// TwinCAT 3 PLC project CNM_AssertionInterfaceLib
// Title: CNM_AssertionInterfaces
// Company: ekvip automation GmbH
// Author: elfrosch
// ProjectVersion: 0.1.1.0
// Description: This library provides an abstract class `AbstractAssertor` to ease assert statements. It provides assert statements in a [fluent interface](https://en.wikipedia.org/wiki/Fluent_interface) style for the most common data types. .. <legal notes> legal notes ================= | SPDX-FileCopyrightText: © 2022 ekvip automation GmbH <info@ekvip.de> | SPDX-License-Identifier: Apache-2.0 | For details check: Apache-2.0_ .. _Apache-2.0: https://www.apache.org/licenses/LICENSE-2.0 .. </legal notes>
// ProgramVersion: 3.1.4026.19
// libraries:
//   CNM_AbstractObject, * (ekvip automation GmbH)
//   CNM_ReturnTypes, * (ekvip automation GmbH)
//   CNM_UnicodeUtilities, * (ekvip automation GmbH)
//   SysMem, * (System)
//   Tc2_Standard, * (Beckhoff Automation GmbH)
//   Tc2_System, * (Beckhoff Automation GmbH)
//   Tc2_Utilities, * (Beckhoff Automation GmbH)
// project tree:
//   Assertor/Assertions/BinaryAssertions/classes/ BinaryAssertions.TcPOU
//   Assertor/Assertions/BinaryAssertions/interfaces/ IBinaryAssertions.TcIO
//   Assertor/Assertions/BitNumberAssertions/Byte/classes/ ByteAssertions.TcPOU
//   Assertor/Assertions/BitNumberAssertions/Byte/interfaces/ IByteAssertions.TcIO
//   Assertor/Assertions/BitNumberAssertions/Byte/types/subranges/ BitNumberByte.TcDUT
//   Assertor/Assertions/BitNumberAssertions/classes/ BitNumberAssertions.TcPOU
//   Assertor/Assertions/BitNumberAssertions/Dword/classes/ DWordAssertions.TcPOU
//   Assertor/Assertions/BitNumberAssertions/Dword/interfaces/ IDwordAssertions.TcIO
//   Assertor/Assertions/BitNumberAssertions/Dword/types/subranges/ BitNumberDWord.TcDUT
//   Assertor/Assertions/BitNumberAssertions/interfaces/ IBitNumberAssertions.TcIO
//   Assertor/Assertions/BitNumberAssertions/Lword/classes/ LWordAssertions.TcPOU
//   Assertor/Assertions/BitNumberAssertions/Lword/interfaces/ ILwordAssertions.TcIO
//   Assertor/Assertions/BitNumberAssertions/Lword/types/subranges/ BitNumberLWord.TcDUT
//   Assertor/Assertions/BitNumberAssertions/Word/classes/ WordAssertions.TcPOU
//   Assertor/Assertions/BitNumberAssertions/Word/interfaces/ IWordAssertions.TcIO
//   Assertor/Assertions/BitNumberAssertions/Word/types/subranges/ BitNumberWord.TcDUT
//   Assertor/Assertions/BitNumberAssertions/XWord/classes/ XWordAssertions.TcPOU
//   Assertor/Assertions/BitNumberAssertions/XWord/interfaces/ IXWordAssertions.TcIO
//   Assertor/Assertions/BitNumberAssertions/XWord/types/subranges/ BitNumberXWord.TcDUT
//   Assertor/Assertions/BooleanAssertion/classes/ BooleanAssertion.TcPOU
//   Assertor/Assertions/BooleanAssertion/interfaces/ IBooleanAssertion.TcIO
//   Assertor/Assertions/classes/ Assertions.TcPOU
//   Assertor/Assertions/DateAndTimeAssertions/32Bit/classes/ SimpleDateAndTimeAssertions.TcPOU
//   Assertor/Assertions/DateAndTimeAssertions/32Bit/Date/classes/ DateAssertions32Bit.TcPOU
//   Assertor/Assertions/DateAndTimeAssertions/32Bit/Date/interfaces/ I32BitDateAssertions.TcIO
//   Assertor/Assertions/DateAndTimeAssertions/32Bit/DT/classes/ DateTimeAssertions32Bit.TcPOU
//   Assertor/Assertions/DateAndTimeAssertions/32Bit/DT/interfaces/ I32BitDtAssertions.TcIO
//   Assertor/Assertions/DateAndTimeAssertions/32Bit/interfaces/ ISimpleDateAndTimeAssertions.TcIO
//   Assertor/Assertions/DateAndTimeAssertions/32Bit/TOD/classes/ TimeOfDayAssertions32Bit.TcPOU
//   Assertor/Assertions/DateAndTimeAssertions/32Bit/TOD/interfaces/ I32BitTodAssertions.TcIO
//   Assertor/Assertions/DateAndTimeAssertions/64Bit/classes/ LongDateAndTimeAssertions.TcPOU
//   Assertor/Assertions/DateAndTimeAssertions/64Bit/LDate/classes/ DateAssertions64Bit.TcPOU
//   Assertor/Assertions/DateAndTimeAssertions/64Bit/LDate/interfaces/ I64BitDateAssertions.TcIO
//   Assertor/Assertions/DateAndTimeAssertions/64Bit/LDT/classes/ DateTimeAssertions64Bit.TcPOU
//   Assertor/Assertions/DateAndTimeAssertions/64Bit/LDT/interfaces/ I64BitDtAssertions.TcIO
//   Assertor/Assertions/DateAndTimeAssertions/64Bit/interfaces/ ILongDateAndTimeAssertions.TcIO
//   Assertor/Assertions/DateAndTimeAssertions/64Bit/LTOD/classes/ TimeOfDayAssertions64Bit.TcPOU
//   Assertor/Assertions/DateAndTimeAssertions/64Bit/LTOD/interfaces/ I64BitTodAssertions.TcIO
//   Assertor/Assertions/DateAndTimeAssertions/classes/ DateAndTimeAssertions.TcPOU
//   Assertor/Assertions/DateAndTimeAssertions/interfaces/ IDateAndTimeAssertions.TcIO
//   Assertor/Assertions/FloatAssertions/classes/ FloatAssertions.TcPOU
//   Assertor/Assertions/FloatAssertions/interfaces/ IFloatAssertions.TcIO
//   Assertor/Assertions/FloatAssertions/Lreal/classes/ LrealAssertions.TcPOU
//   Assertor/Assertions/FloatAssertions/Lreal/interfaces/ ILrealAssertions.TcIO
//   Assertor/Assertions/FloatAssertions/Real/classes/ RealAssertions.TcPOU
//   Assertor/Assertions/FloatAssertions/Real/interfaces/ IRealAssertions.TcIO
//   Assertor/Assertions/IntegerAssertions/classes/ IntegerAssertions.TcPOU
//   Assertor/Assertions/IntegerAssertions/interfaces/ IIntegerAssertions.TcIO
//   Assertor/Assertions/IntegerAssertions/signed/classes/ SignedIntegerAssertions.TcPOU
//   Assertor/Assertions/IntegerAssertions/signed/Dint/classes/ DintAssertions.TcPOU
//   Assertor/Assertions/IntegerAssertions/signed/Dint/interfaces/ IDintAssertions.TcIO
//   Assertor/Assertions/IntegerAssertions/signed/interfaces/ ISignedIntegerAssertions.TcIO
//   Assertor/Assertions/IntegerAssertions/signed/Int/classes/ IntAssertions.TcPOU
//   Assertor/Assertions/IntegerAssertions/signed/Int/interfaces/ IIntAssertions.TcIO
//   Assertor/Assertions/IntegerAssertions/signed/Lint/classes/ LintAssertions.TcPOU
//   Assertor/Assertions/IntegerAssertions/signed/Lint/interfaces/ ILintAssertions.TcIO
//   Assertor/Assertions/IntegerAssertions/signed/Sint/classes/ SintAssertions.TcPOU
//   Assertor/Assertions/IntegerAssertions/signed/Sint/interfaces/ ISintAssertions.TcIO
//   Assertor/Assertions/IntegerAssertions/signed/Xint/classes/ XintAssertions.TcPOU
//   Assertor/Assertions/IntegerAssertions/signed/Xint/interfaces/ IXintAssertions.TcIO
//   Assertor/Assertions/IntegerAssertions/unsigned/classes/ UnsignedIntegerAssertions.TcPOU
//   Assertor/Assertions/IntegerAssertions/unsigned/interfaces/ IUnsignedIntegerAssertions.TcIO
//   Assertor/Assertions/IntegerAssertions/unsigned/Udint/classes/ UdintAssertions.TcPOU
//   Assertor/Assertions/IntegerAssertions/unsigned/Udint/interfaces/ IUdintAssertions.TcIO
//   Assertor/Assertions/IntegerAssertions/unsigned/Uint/classes/ UintAssertions.TcPOU
//   Assertor/Assertions/IntegerAssertions/unsigned/Uint/interfaces/ IUintAssertions.TcIO
//   Assertor/Assertions/IntegerAssertions/unsigned/Ulint/classes/ UlintAssertions.TcPOU
//   Assertor/Assertions/IntegerAssertions/unsigned/Ulint/interfaces/ IUlintAssertions.TcIO
//   Assertor/Assertions/IntegerAssertions/unsigned/Usint/classes/ UsintAssertions.TcPOU
//   Assertor/Assertions/IntegerAssertions/unsigned/Usint/interfaces/ IUsintAssertions.TcIO
//   Assertor/Assertions/IntegerAssertions/unsigned/Uxint/classes/ UxintAssertions.TcPOU
//   Assertor/Assertions/IntegerAssertions/unsigned/Uxint/interfaces/ IUxintAssertions.TcIO
//   Assertor/Assertions/interfaces/ IAssertions.TcIO
//   Assertor/Assertions/ObjectAssertions/classes/ ObjectAssertions.TcPOU
//   Assertor/Assertions/ObjectAssertions/interfaces/ IObjectAssertions.TcIO
//   Assertor/Assertions/PointerAssertions/classes/ PointerAssertions.TcPOU
//   Assertor/Assertions/PointerAssertions/interfaces/ IPointerAssertions.TcIO
//   Assertor/Assertions/StringAssertion/classes/ AbstractStringPointerAssertions.TcPOU, StringAssertions.TcPOU
//   Assertor/Assertions/StringAssertion/interfaces/ IStringAssertions.TcIO
//   Assertor/Assertions/StringAssertion/Win125x/classes/ Windows125xStringAssertions.TcPOU, Windows125xStringPointerAssertions.TcPOU
//   Assertor/Assertions/StringAssertion/Win125x/interfaces/ IWindows125xStringAssertions.TcIO, IWindows125xStringPointerAssertions.TcIO
//   Assertor/Assertions/StringAssertion/Unicode/Classes/ UnicodeAssertions.TcPOU
//   Assertor/Assertions/StringAssertion/Unicode/Classes/UTF-16/ Utf16StringAssertions.TcPOU, Utf16StringPointerAssertions.TcPOU
//   Assertor/Assertions/StringAssertion/Unicode/Classes/UTF-8/ Utf8StringAssertions.TcPOU, Utf8StringPointerAssertions.TcPOU
//   Assertor/Assertions/StringAssertion/Unicode/enumerations/ UnicodeStringLengthUnit.TcDUT
//   Assertor/Assertions/StringAssertion/Unicode/Interfaces/ IUnicodeStringAssertions.TcIO
//   Assertor/Assertions/StringAssertion/Unicode/Interfaces/UTF-16/ IUtf16StringAssertions.TcIO, IUtf16StringPointerAssertions.TcIO
//   Assertor/Assertions/StringAssertion/Unicode/Interfaces/UTF-8/ IUtf8StringAssertions.TcIO, IUtf8StringPointerAssertions.TcIO
//   Assertor/Assertions/TimeAssertions/classes/ TimeAssertions.TcPOU
//   Assertor/Assertions/TimeAssertions/interfaces/ ITimeAssertions.TcIO
//   Assertor/Assertions/TimeAssertions/LTime/classes/ LongTimeAssertions.TcPOU
//   Assertor/Assertions/TimeAssertions/LTime/interfaces/ I64BitTimeAssertions.TcIO
//   Assertor/Assertions/TimeAssertions/Time/classes/ SimpleTimeAssertions.TcPOU
//   Assertor/Assertions/TimeAssertions/Time/interfaces/ I32BitTimeAssertions.TcIO
//   Assertor/classes/ AbstractAssertion.TcPOU, AbstractAssertor.TcPOU
//   Assertor/interfaces/ IAssertor.TcIO, IAssertCallBack.TcIO, IAssertCallBackSetter.TcIO
//   Assertor/types/aliases/ AssertMessage.TcDUT
//   Project Information/ F_GetCompany.TcPOU, F_GetTitle.TcPOU, F_GetVersion.TcPOU
//   Version/ Global_Version.TcGVL
// real-time tasks:
//   TASK CNC-Task ADS: cycle default, priority 7, ADS port 558
//   TASK CNC-Task COM: cycle T#10ms, priority 13, ADS port 556
//   TASK CNC-Task SDA: cycle T#10ms, priority 8, ADS port 555
//   TASK CNC-Task GEO: cycle T#2ms, priority 3, ADS port 554

// ---- Assertor/Assertions/BitNumberAssertions/Byte/types/subranges/BitNumberByte.TcDUT
(*

## Short summary

BitNumberByte is an alias of ``USINT(0..7)``.
This data type exists so that no one can provoke an overflow of the bit numbers.
It's used as parameter at 
`IByteAssertions.bitXIsEqualTo` 
`IByteAssertions.bitXIsNotEqualTo` 
`IByteAssertions.bitXIsSet` 
`IByteAssertions.bitXIsUnset` 

.. <legal notes>

legal notes
=================
| SPDX-FileCopyrightText: © 2022 ekvip automation GmbH <info@ekvip.de>
| SPDX-License-Identifier: Apache-2.0
| For details check: Apache-2.0_

.. _Apache-2.0: https://www.apache.org/licenses/LICENSE-2.0

.. </legal notes>

*)

TYPE
	BitNumberByte :USINT(0..7); 
END_TYPE

// ---- Assertor/Assertions/BitNumberAssertions/Dword/types/subranges/BitNumberDWord.TcDUT
(*

## Short summary

 BitNumberDWord is an alias of ``USINT(0..31)``.
 This data type exists so that no one can provoke an overflow of the bit numbers.
 It's used as parameter of 
 `IDwordAssertions.bitXIsEqualTo` 
 `IDwordAssertions.bitXIsNotEqualTo` 
 `IDwordAssertions.bitXIsSet` 
 `IDwordAssertions.bitXIsUnset` 

.. <legal notes>

legal notes
=================
| SPDX-FileCopyrightText: © 2022 ekvip automation GmbH <info@ekvip.de>
| SPDX-License-Identifier: Apache-2.0
| For details check: Apache-2.0_

.. _Apache-2.0: https://www.apache.org/licenses/LICENSE-2.0

.. </legal notes>

*)

TYPE
	BitNumberDWord :USINT(0..31);
END_TYPE

// ---- Assertor/Assertions/BitNumberAssertions/Lword/types/subranges/BitNumberLWord.TcDUT
(*

## Short summary

BitNumberLWord is an alias of ``USINT(0..63)``.
This data type exists so that no one can provoke an overflow of the bit numbers.
It's used as parameter of 
`ILwordAssertions.bitXIsEqualTo` 
`ILwordAssertions.bitXIsNotEqualTo` 
`ILwordAssertions.bitXIsSet` 
`ILwordAssertions.bitXIsUnset` 

.. <legal notes>

legal notes
=================
| SPDX-FileCopyrightText: © 2022 ekvip automation GmbH <info@ekvip.de>
| SPDX-License-Identifier: Apache-2.0
| For details check: Apache-2.0_

.. _Apache-2.0: https://www.apache.org/licenses/LICENSE-2.0

.. </legal notes>

*)

TYPE
	BitNumberLWord :USINT(0..63);
END_TYPE

// ---- Assertor/Assertions/BitNumberAssertions/Word/types/subranges/BitNumberWord.TcDUT
(*

## Short summary

BitNumberWord is an alias of ``USINT(0..15)``.
This data type exists so that no one can provoke an overflow of the bit numbers.
It's used as parameter of 
`IWordAssertions.bitXIsEqualTo` 
`IWordAssertions.bitXIsNotEqualTo` 
`IWordAssertions.bitXIsSet` 
`IWordAssertions.bitXIsUnset` 

.. <legal notes>

legal notes
=================
| SPDX-FileCopyrightText: © 2022 ekvip automation GmbH <info@ekvip.de>
| SPDX-License-Identifier: Apache-2.0
| For details check: Apache-2.0_

.. _Apache-2.0: https://www.apache.org/licenses/LICENSE-2.0

.. </legal notes>

*)

TYPE
	BitNumberWord :USINT(0..15);
END_TYPE

// ---- Assertor/Assertions/BitNumberAssertions/XWord/types/subranges/BitNumberXWord.TcDUT
(*

## Short summary

BitNumberXWord is
for 32 bit machines an alias of ``USINT(0..31)``
for 64 bit machines an alias of ``USINT(0..63)``
This data type exists so that no one can provoke an overflow of the bit numbers.
It's used as parameter of 
`IXWordAssertions.bitXIsEqualTo` 
`IXWordAssertions.bitXIsNotEqualTo` 
`IXWordAssertions.bitXIsSet` 
`IXWordAssertions.bitXIsUnset` 

.. <legal notes>

legal notes
=================
| SPDX-FileCopyrightText: © 2022 ekvip automation GmbH <info@ekvip.de>
| SPDX-License-Identifier: Apache-2.0
| For details check: Apache-2.0_

.. _Apache-2.0: https://www.apache.org/licenses/LICENSE-2.0

.. </legal notes>

*)

TYPE
	BitNumberXWord :USINT(0..((SIZEOF(__XWORD)*8)-1));
END_TYPE

// ---- Assertor/Assertions/StringAssertion/Unicode/enumerations/UnicodeStringLengthUnit.TcDUT
(*

## Short summary
This list is intended to define the string length units of measurement

Type of the enumartion is ``BYTE``

.. <legal notes>

legal notes
=================
| SPDX-FileCopyrightText: © 2022 ekvip automation GmbH <info@ekvip.de>
| SPDX-License-Identifier: Apache-2.0
| For details check: Apache-2.0_

.. _Apache-2.0: https://www.apache.org/licenses/LICENSE-2.0

.. </legal notes>

enumeration values
======================

*)

{attribute 'qualified_only'}
{attribute 'strict'}
{attribute 'to_string'}
TYPE UnicodeStringLengthUnit :
(
	(* Just the number of bytes without the termination character U+0000 *)
	BYTES := 0,
	(* 
	Character count of a string. For example Ä
	can be represented just one character U+00C4 (Ä) 
	or it can be represented by two characters U+0041 U+00308 (A◌̈)
	*)
	CHARACTERS := 1,
	(*
	Character count of a string normalized with form D.
	Form D is a canonical decomposition. 
	For example Ä (U+00C4) will transformed to A◌̈ (U+0041 U+00308)
	both count as two in NFD.
	*)
	CHARACTERS_NFD := 2,
	(*
	Character count of a string normalized with form C.
	Form C is a canonial composition. 
	For example A◌̈ (U+0041 U+00308) will transformed to Ä (U+00C4)
	both count as one in NFC.
	*)	
	CHARACTERS_NFC := 3,
	(*
	Character count of a string but the visible only.
	For example the developer emoji 👨‍💻 is made from three characters:
	man👨 (U+1F468),zero width joiner (U+200D) and the Personal Computer 💻 (U+1F4BB)
	but it counts just one for it.
	*)
	VISIBLE_CHARACTERS := 4,
	(*
	String width (rendering width according to the number of spaces (U+0020)).
 	If strings should be horizontally aligned, then it's required to check the width.
	For example woman 👩 (U+1F469) has a width of two spaces, 
	developer 👨‍💻 (U+1F468 U+200D U+1F4BB) has a width of five spaces
	and Ä has a width of one space
	*)
	WIDTH := 5
)DINT;
END_TYPE

// ---- Assertor/types/aliases/AssertMessage.TcDUT
(*

## Short summary
AssertMessage is an alias of Tc2_System.T_MaxString.
It's just a tmeporary type to ease the change to 
an alarm event (but there is no library for this yet)

.. <legal notes>

legal notes
=================
| SPDX-FileCopyrightText: © 2022 ekvip automation GmbH <info@ekvip.de>
| SPDX-License-Identifier: Apache-2.0
| For details check: Apache-2.0_

.. _Apache-2.0: https://www.apache.org/licenses/LICENSE-2.0

.. </legal notes>

*)

TYPE
	AssertMessage :Tc2_System.T_MaxString;
END_TYPE

// ---- Version/Global_Version.TcGVL
{attribute 'TcGenerated'}
{attribute 'no-analysis'}
{attribute 'linkalways'}
// This function has been automatically generated from the project information.
VAR_GLOBAL CONSTANT
	{attribute 'const_non_replaced'}
	stLibVersion_CNM_AssertionInterfaces : ST_LibVersion := (iMajor := 0, iMinor := 1, iBuild := 1, iRevision := 0, nFlags := 0, sVersion := '0.1.1.0');
END_VAR

// ---- Assertor/Assertions/BinaryAssertions/interfaces/IBinaryAssertions.TcIO
(*

## Short summary
This interface provides assert statements for binaries
e.g. structures, arrays etc...  

.. <legal notes>

legal notes
=================
| SPDX-FileCopyrightText: © 2022 ekvip automation GmbH <info@ekvip.de>
| SPDX-License-Identifier: Apache-2.0
| For details check: Apache-2.0_

.. _Apache-2.0: https://www.apache.org/licenses/LICENSE-2.0

.. </legal notes>



*)

INTERFACE IBinaryAssertions EXTENDS __SYSTEM.IQueryInterface

(*

## Short summary
This assertion method checks if all bytes of memory of
``data`` and ``dataToCompare`` are equal

**Attention:** 
	Binary comparison means it compares values byte by byte, regardless of type information (signs, ``REAL`` etc...)
	and it compares padding bytes, too.

**Attention:** 
	``STRING`` and ``WSTRING`` is null terminated
	that means TwinCAT sets null byte/word at the end of the string and touches nothing else
	For example ``foo :STRING(3) := 'foo';`` looks binary 16#66 16#6F 16#6F 16#00.
	if you set foo to an empty string ``foo := ''`` it looks like 16#00 16#6F 16#6F 16#00.

.. <legal notes>

legal notes
=================
| SPDX-FileCopyrightText: © 2022 ekvip automation GmbH <info@ekvip.de>
| SPDX-License-Identifier: Apache-2.0
| For details check: Apache-2.0_

.. _Apache-2.0: https://www.apache.org/licenses/LICENSE-2.0

.. </legal notes>



*)

METHOD isEqualTo
VAR_INPUT
	(* current binary data *)
	data			:ANY;
	(* binary data with the expected values *)
	dataToCompare	:ANY;
	(* message if the assertion is false *)
	message			:AssertMessage;
END_VAR
END_METHOD

(*

## Short summary
This assertion method checks the bytes of memory of
``data`` and ``dataToCompare`` if the content of the first unequal
``data`` byte is greater than the byte of ``dataToCompare``
the assertion is true

**Attention:** 
	Binary comparison means it compares values byte by byte, regardless of type information (signs, ``REAL`` etc...)
	and it compares padding bytes, too.

**Attention:** 
	``STRING`` and ``WSTRING`` is null terminated
	that means TwinCAT sets null byte/word at the end of the string and touches nothing else
	For example ``foo :STRING(3) := 'foo';`` looks binary 16#66 16#6F 16#6F 16#00.
	if you set foo to an empty string ``foo := ''`` it looks like 16#00 16#6F 16#6F 16#00.

.. <legal notes>

legal notes
=================
| SPDX-FileCopyrightText: © 2022 ekvip automation GmbH <info@ekvip.de>
| SPDX-License-Identifier: Apache-2.0
| For details check: Apache-2.0_

.. _Apache-2.0: https://www.apache.org/licenses/LICENSE-2.0

.. </legal notes>



*)

METHOD isGreaterThan
VAR_INPUT
	(* current binary data *)
	data			:ANY;
	(* binary data with smaller values *)
	dataToCompare	:ANY;
	(* message if the assertion is false *)
	message			:AssertMessage;
END_VAR
END_METHOD

(*

## Short summary
This assertion method checks the bytes of memory of
``data`` and ``dataToCompare`` if the content of the first unequal
``data`` byte is less than the byte of ``dataToCompare``
the assertion is true

**Attention:** 
	Binary comparison means it compares values byte by byte, regardless of type information (signs, ``REAL`` etc...)
	and it compares padding bytes, too.

**Attention:** 
	``STRING`` and ``WSTRING`` is null terminated
	that means TwinCAT sets null byte/word at the end of the string and touches nothing else
	For example ``foo :STRING(3) := 'foo';`` looks binary 16#66 16#6F 16#6F 16#00.
	if you set foo to an empty string ``foo := ''`` it looks like 16#00 16#6F 16#6F 16#00.

.. <legal notes>

legal notes
=================
| SPDX-FileCopyrightText: © 2022 ekvip automation GmbH <info@ekvip.de>
| SPDX-License-Identifier: Apache-2.0
| For details check: Apache-2.0_

.. _Apache-2.0: https://www.apache.org/licenses/LICENSE-2.0

.. </legal notes>



*)

METHOD isLessThan
VAR_INPUT
	(* current binary data *)
	data			:ANY;
	(* binary data with greater values *)
	dataToCompare	:ANY;
	(* message if the assertion is false *)
	message			:AssertMessage;
END_VAR
END_METHOD

(*

## Short summary
This assertion method checks if minimal one byte of memory of
``data`` and ``dataToCompare`` is not equal

**Attention:** 
	Binary comparison means it compares values byte by byte, regardless of type information (signs, ``REAL`` etc...)
	and it compares padding bytes, too.

**Attention:** 
	``STRING`` and ``WSTRING`` is null terminated
	that means TwinCAT sets null byte/word at the end of the string and touches nothing else
	For example ``foo :STRING(3) := 'foo';`` looks binary 16#66 16#6F 16#6F 16#00.
	if you set foo to an empty string ``foo := ''`` it looks like 16#00 16#6F 16#6F 16#00.

.. <legal notes>

legal notes
=================
| SPDX-FileCopyrightText: © 2022 ekvip automation GmbH <info@ekvip.de>
| SPDX-License-Identifier: Apache-2.0
| For details check: Apache-2.0_

.. _Apache-2.0: https://www.apache.org/licenses/LICENSE-2.0

.. </legal notes>



*)

METHOD isNotEqualTo
VAR_INPUT
	(* current binary data *)
	data			:ANY;
	(* binary data with the unexpected values *)
	dataToCompare	:ANY;
	(* message if the assertion is false *)
	message			:AssertMessage;
END_VAR
END_METHOD

END_INTERFACE

// ---- Assertor/Assertions/BitNumberAssertions/Byte/interfaces/IByteAssertions.TcIO
(*

## Short summary
This interface provides assert statements for bytes  

.. <legal notes>

legal notes
=================
| SPDX-FileCopyrightText: © 2022 ekvip automation GmbH <info@ekvip.de>
| SPDX-License-Identifier: Apache-2.0
| For details check: Apache-2.0_

.. _Apache-2.0: https://www.apache.org/licenses/LICENSE-2.0

.. </legal notes>



*)

INTERFACE IByteAssertions EXTENDS __SYSTEM.IQueryInterface

(*

## Short summary
This assertion method checks if the result current value bitwise ``AND`` mask is equal to the expected value

.. <legal notes>

legal notes
=================
| SPDX-FileCopyrightText: © 2022 ekvip automation GmbH <info@ekvip.de>
| SPDX-License-Identifier: Apache-2.0
| For details check: Apache-2.0_

.. _Apache-2.0: https://www.apache.org/licenses/LICENSE-2.0

.. </legal notes>



*)

METHOD andMaskIsEqualTo
VAR_INPUT
	(* current value to check *)
	currentValue	:BYTE;
	(* 2nd operand for bitwise operation *)
	mask			:BYTE;
	(* expected result after masking *)
	expectedValue	:BYTE;
	(* message if the assertion is false *)
	message			:AssertMessage;
END_VAR
END_METHOD

(*

## Short summary
This assertion method checks if the result current value bitwise ``AND`` mask
is not equal to the unexpected value

.. <legal notes>

legal notes
=================
| SPDX-FileCopyrightText: © 2022 ekvip automation GmbH <info@ekvip.de>
| SPDX-License-Identifier: Apache-2.0
| For details check: Apache-2.0_

.. _Apache-2.0: https://www.apache.org/licenses/LICENSE-2.0

.. </legal notes>



*)

METHOD andMaskIsNotEqualTo
VAR_INPUT
	(* current value to check *)
	currentValue	:BYTE;
	(* 2nd operand for bitwise operation *)
	mask			:BYTE;
	(* unexpected result after masking *)
	unexpectedValue	:BYTE;
	(* message if the assertion is false *)
	message			:AssertMessage;
END_VAR
END_METHOD

(*

## Short summary
This assertion method checks if the selected bit of current value
is equal to the expected value

.. <legal notes>

legal notes
=================
| SPDX-FileCopyrightText: © 2022 ekvip automation GmbH <info@ekvip.de>
| SPDX-License-Identifier: Apache-2.0
| For details check: Apache-2.0_

.. _Apache-2.0: https://www.apache.org/licenses/LICENSE-2.0

.. </legal notes>



*)

METHOD bitXIsEqualTo
VAR_INPUT
	(* current value to check *)
	currentValue	:BYTE;
	(* number of bit to check *)
	number			:BitNumberByte;	
	(* expected value of bit *)
	expectedValue	:BOOL;
	(* message if the assertion is false *)
	message			:AssertMessage;
END_VAR
END_METHOD

(*

## Short summary
This assertion method checks if the selected bit of current value
is not equal to the unexpected value

.. <legal notes>

legal notes
=================
| SPDX-FileCopyrightText: © 2022 ekvip automation GmbH <info@ekvip.de>
| SPDX-License-Identifier: Apache-2.0
| For details check: Apache-2.0_

.. _Apache-2.0: https://www.apache.org/licenses/LICENSE-2.0

.. </legal notes>



*)

METHOD bitXIsNotEqualTo
VAR_INPUT
	(* current value to check *)
	currentValue	:BYTE;
	(* number of bit to check *)
	number			:BitNumberByte;	
	(* unexpected value of bit *)
	unexpectedValue	:BOOL;
	(* message if the assertion is false *)
	message			:AssertMessage;
END_VAR
END_METHOD

(*

## Short summary
This assertion method checks if the selected bit of current value
is set

.. <legal notes>

legal notes
=================
| SPDX-FileCopyrightText: © 2022 ekvip automation GmbH <info@ekvip.de>
| SPDX-License-Identifier: Apache-2.0
| For details check: Apache-2.0_

.. _Apache-2.0: https://www.apache.org/licenses/LICENSE-2.0

.. </legal notes>



*)

METHOD bitXIsSet
VAR_INPUT
	(* current value to check *)
	currentValue	:BYTE;
	(* number of bit to check *)
	number			:BitNumberByte;	
	(* message if the assertion is false *)
	message			:AssertMessage;
END_VAR
END_METHOD

(*

## Short summary
This assertion method checks if the selected bit of current value
is unset

.. <legal notes>

legal notes
=================
| SPDX-FileCopyrightText: © 2022 ekvip automation GmbH <info@ekvip.de>
| SPDX-License-Identifier: Apache-2.0
| For details check: Apache-2.0_

.. _Apache-2.0: https://www.apache.org/licenses/LICENSE-2.0

.. </legal notes>



*)

METHOD bitXIsUnset
VAR_INPUT
	(* current value to check *)
	currentValue	:BYTE;
	(* number of bit to check *)
	number			:BitNumberByte;	
	(* message if the assertion is false *)
	message			:AssertMessage;
END_VAR
END_METHOD

(*

## Short summary
This assertion method checks if the least significant bit of current value
is equal to the expected value

.. <legal notes>

legal notes
=================
| SPDX-FileCopyrightText: © 2022 ekvip automation GmbH <info@ekvip.de>
| SPDX-License-Identifier: Apache-2.0
| For details check: Apache-2.0_

.. _Apache-2.0: https://www.apache.org/licenses/LICENSE-2.0

.. </legal notes>



*)

METHOD lsbIsEqualTo
VAR_INPUT
	(* current value to check *)
	currentValue	:BYTE;
	(* expected value of lsb *)
	expectedValue	:BOOL;
	(* message if the assertion is false *)
	message			:AssertMessage;
END_VAR
END_METHOD

(*

## Short summary
This assertion method checks if the least significant bit of current value
is not equal to the unexpected value

.. <legal notes>

legal notes
=================
| SPDX-FileCopyrightText: © 2022 ekvip automation GmbH <info@ekvip.de>
| SPDX-License-Identifier: Apache-2.0
| For details check: Apache-2.0_

.. _Apache-2.0: https://www.apache.org/licenses/LICENSE-2.0

.. </legal notes>



*)

METHOD lsbIsNotEqualTo
VAR_INPUT
	(* current value to check *)
	currentValue	:BYTE;
	(* unexpected value of lsb *)
	unexpectedValue	:BOOL;
	(* message if the assertion is false *)
	message			:AssertMessage;
END_VAR
END_METHOD

(*

## Short summary
This assertion method checks if the least significant bit of current value
is set

.. <legal notes>

legal notes
=================
| SPDX-FileCopyrightText: © 2022 ekvip automation GmbH <info@ekvip.de>
| SPDX-License-Identifier: Apache-2.0
| For details check: Apache-2.0_

.. _Apache-2.0: https://www.apache.org/licenses/LICENSE-2.0

.. </legal notes>



*)

METHOD lsbIsSet
VAR_INPUT
	(* current value to check *)
	currentValue	:BYTE;
	(* message if the assertion is false *)
	message			:AssertMessage;
END_VAR
END_METHOD

(*

## Short summary
This assertion method checks if the least significant bit of current value
is unset

.. <legal notes>

legal notes
=================
| SPDX-FileCopyrightText: © 2022 ekvip automation GmbH <info@ekvip.de>
| SPDX-License-Identifier: Apache-2.0
| For details check: Apache-2.0_

.. _Apache-2.0: https://www.apache.org/licenses/LICENSE-2.0

.. </legal notes>



*)

METHOD lsbIsUnset
VAR_INPUT
	(* current value to check *)
	currentValue	:BYTE;
	(* message if the assertion is false *)
	message			:AssertMessage;
END_VAR
END_METHOD

(*

## Short summary
This assertion method checks if the most significant bit of current value
is equal to the expected value

.. <legal notes>

legal notes
=================
| SPDX-FileCopyrightText: © 2022 ekvip automation GmbH <info@ekvip.de>
| SPDX-License-Identifier: Apache-2.0
| For details check: Apache-2.0_

.. _Apache-2.0: https://www.apache.org/licenses/LICENSE-2.0

.. </legal notes>



*)

METHOD msbIsEqualTo
VAR_INPUT
	(* current value to check *)
	currentValue	:BYTE;
	(* expected value of msb *)
	expectedValue	:BOOL;
	(* message if the assertion is false *)
	message			:AssertMessage;
END_VAR
END_METHOD

(*

## Short summary
This assertion method checks if the most significant bit of current value
is not equal to the unexpected value

.. <legal notes>

legal notes
=================
| SPDX-FileCopyrightText: © 2022 ekvip automation GmbH <info@ekvip.de>
| SPDX-License-Identifier: Apache-2.0
| For details check: Apache-2.0_

.. _Apache-2.0: https://www.apache.org/licenses/LICENSE-2.0

.. </legal notes>



*)

METHOD msbIsNotEqualTo
VAR_INPUT
	(* current value to check *)
	currentValue	:BYTE;
	(* unexpected value of msb *)
	unexpectedValue	:BOOL;
	(* message if the assertion is false *)
	message			:AssertMessage;
END_VAR
END_METHOD

(*

## Short summary
This assertion method checks if the most significant bit of current value
is set

.. <legal notes>

legal notes
=================
| SPDX-FileCopyrightText: © 2022 ekvip automation GmbH <info@ekvip.de>
| SPDX-License-Identifier: Apache-2.0
| For details check: Apache-2.0_

.. _Apache-2.0: https://www.apache.org/licenses/LICENSE-2.0

.. </legal notes>



*)

METHOD msbIsSet
VAR_INPUT
	(* current value to check *)
	currentValue	:BYTE;
	(* message if the assertion is false *)
	message			:AssertMessage;
END_VAR
END_METHOD

(*

## Short summary
This assertion method checks if the most significant bit of current value
is unset

.. <legal notes>

legal notes
=================
| SPDX-FileCopyrightText: © 2022 ekvip automation GmbH <info@ekvip.de>
| SPDX-License-Identifier: Apache-2.0
| For details check: Apache-2.0_

.. _Apache-2.0: https://www.apache.org/licenses/LICENSE-2.0

.. </legal notes>



*)

METHOD msbIsUnset
VAR_INPUT
	(* current value to check *)
	currentValue	:BYTE;
	(* message if the assertion is false *)
	message			:AssertMessage;
END_VAR
END_METHOD

(*

## Short summary
This assertion method checks if the result current value bitwise ``OR`` mask is equal to the expected value

.. <legal notes>

legal notes
=================
| SPDX-FileCopyrightText: © 2022 ekvip automation GmbH <info@ekvip.de>
| SPDX-License-Identifier: Apache-2.0
| For details check: Apache-2.0_

.. _Apache-2.0: https://www.apache.org/licenses/LICENSE-2.0

.. </legal notes>



*)

METHOD orMaskIsEqualTo
VAR_INPUT
	(* current value to check *)
	currentValue	:BYTE;
	(* 2nd operand for bitwise operation *)
	mask			:BYTE;
	(* expected result after masking *)
	expectedValue	:BYTE;
	(* message if the assertion is false *)
	message			:AssertMessage;
END_VAR
END_METHOD

(*

## Short summary
This assertion method checks if the result current value bitwise ``OR`` mask 
is not equal to the unexpected value

.. <legal notes>

legal notes
=================
| SPDX-FileCopyrightText: © 2022 ekvip automation GmbH <info@ekvip.de>
| SPDX-License-Identifier: Apache-2.0
| For details check: Apache-2.0_

.. _Apache-2.0: https://www.apache.org/licenses/LICENSE-2.0

.. </legal notes>



*)

METHOD orMaskIsNotEqualTo
VAR_INPUT
	(* current value to check *)
	currentValue	:BYTE;
	(* 2nd operand for bitwise operation *)
	mask			:BYTE;
	(* unexpected result after masking *)
	unexpectedValue	:BYTE;
	(* message if the assertion is false *)
	message			:AssertMessage;
END_VAR
END_METHOD

(*

## Short summary
This assertion method checks if the current value is equal to the expected value

.. <legal notes>

legal notes
=================
| SPDX-FileCopyrightText: © 2022 ekvip automation GmbH <info@ekvip.de>
| SPDX-License-Identifier: Apache-2.0
| For details check: Apache-2.0_

.. _Apache-2.0: https://www.apache.org/licenses/LICENSE-2.0

.. </legal notes>



*)

METHOD valueIsEqualTo
VAR_INPUT
	(* current value to check *)
	currentValue	:BYTE;
	(* expected value to compare *)
	expectedValue	:BYTE;
	(* message if the assertion is false *)
	message			:AssertMessage;
END_VAR
END_METHOD

(*

## Short summary
This assertion method checks if the current value is greater than the less value

.. <legal notes>

legal notes
=================
| SPDX-FileCopyrightText: © 2022 ekvip automation GmbH <info@ekvip.de>
| SPDX-License-Identifier: Apache-2.0
| For details check: Apache-2.0_

.. _Apache-2.0: https://www.apache.org/licenses/LICENSE-2.0

.. </legal notes>



*)

METHOD valueIsGreaterThan
VAR_INPUT
	(* current value to check *)
	currentValue	:BYTE;
	(* less than lower limit *)
	lessValue		:BYTE;
	(* message if the assertion is false *)
	message			:AssertMessage;
END_VAR
END_METHOD

(*

## Short summary
This assertion method checks if the current value is inside a limit

**Attention:** 
	limits are included: ``valueIsInRangeOf(3, 3, 3)`` is a true assertion

.. <legal notes>

legal notes
=================
| SPDX-FileCopyrightText: © 2022 ekvip automation GmbH <info@ekvip.de>
| SPDX-License-Identifier: Apache-2.0
| For details check: Apache-2.0_

.. _Apache-2.0: https://www.apache.org/licenses/LICENSE-2.0

.. </legal notes>



*)

METHOD valueIsInRangeOf
VAR_INPUT
	(* lower limit for the current value *)
	lowerLimit		:BYTE;
	(* current value to check *)
	currentValue	:BYTE;
	(* upper limit for the current value *)
	upperLimit		:BYTE;
	(* message if the assertion is false *)
	message			:AssertMessage;
END_VAR
END_METHOD

(*

## Short summary
This assertion method checks if the current value is less than the greater value

.. <legal notes>

legal notes
=================
| SPDX-FileCopyrightText: © 2022 ekvip automation GmbH <info@ekvip.de>
| SPDX-License-Identifier: Apache-2.0
| For details check: Apache-2.0_

.. _Apache-2.0: https://www.apache.org/licenses/LICENSE-2.0

.. </legal notes>



*)

METHOD valueIsLessThan
VAR_INPUT
	(* current value to check *)
	currentValue	:BYTE;
	(* greater than upper limit *)
	greaterValue	:BYTE;
	(* message if the assertion is false *)
	message			:AssertMessage;
END_VAR
END_METHOD

(*

## Short summary
This assertion method checks if the current value is less than or equal to the maximum value

.. <legal notes>

legal notes
=================
| SPDX-FileCopyrightText: © 2022 ekvip automation GmbH <info@ekvip.de>
| SPDX-License-Identifier: Apache-2.0
| For details check: Apache-2.0_

.. _Apache-2.0: https://www.apache.org/licenses/LICENSE-2.0

.. </legal notes>



*)

METHOD valueIsMax
VAR_INPUT
	(* current value to check *)
	currentValue	:BYTE;
	(* upper limit for the current value *)
	maximumValue	:BYTE;
	(* message if the assertion is false *)
	message			:AssertMessage;
END_VAR
END_METHOD

(*

## Short summary
This assertion method checks if the current value is greater than or equal to the minimum value

.. <legal notes>

legal notes
=================
| SPDX-FileCopyrightText: © 2022 ekvip automation GmbH <info@ekvip.de>
| SPDX-License-Identifier: Apache-2.0
| For details check: Apache-2.0_

.. _Apache-2.0: https://www.apache.org/licenses/LICENSE-2.0

.. </legal notes>



*)

METHOD valueIsMin
VAR_INPUT
	(* current value to check *)
	currentValue	:BYTE;
	(* lower limit for the current value *)
	minimumValue	:BYTE;
	(* message if the assertion is false *)
	message			:AssertMessage;
END_VAR
END_METHOD

(*

## Short summary
This assertion method checks if the current value is not equal to the unexpected value

.. <legal notes>

legal notes
=================
| SPDX-FileCopyrightText: © 2022 ekvip automation GmbH <info@ekvip.de>
| SPDX-License-Identifier: Apache-2.0
| For details check: Apache-2.0_

.. _Apache-2.0: https://www.apache.org/licenses/LICENSE-2.0

.. </legal notes>



*)

METHOD valueIsNotEqualTo
VAR_INPUT
	(* current value to check *)
	currentValue	:BYTE;
	(* unexpected value to compare *)
	unexpectedValue	:BYTE;
	(* message if the assertion is false *)
	message			:AssertMessage;
END_VAR
END_METHOD

(*

## Short summary
This assertion method checks if the result current value bitwise ``XOR`` mask is equal to the expected value

.. <legal notes>

legal notes
=================
| SPDX-FileCopyrightText: © 2022 ekvip automation GmbH <info@ekvip.de>
| SPDX-License-Identifier: Apache-2.0
| For details check: Apache-2.0_

.. _Apache-2.0: https://www.apache.org/licenses/LICENSE-2.0

.. </legal notes>



*)

METHOD xorMaskIsEqualTo
VAR_INPUT
	(* current value to check *)
	currentValue	:BYTE;
	(* 2nd operand for bitwise operation *)
	mask			:BYTE;
	(* expected result after masking *)
	expectedValue	:BYTE;
	(* message if the assertion is false *)
	message			:AssertMessage;
END_VAR
END_METHOD

(*

## Short summary
This assertion method checks if the result current value bitwise ``XOR`` mask 
is not equal to the unexpected value

.. <legal notes>

legal notes
=================
| SPDX-FileCopyrightText: © 2022 ekvip automation GmbH <info@ekvip.de>
| SPDX-License-Identifier: Apache-2.0
| For details check: Apache-2.0_

.. _Apache-2.0: https://www.apache.org/licenses/LICENSE-2.0

.. </legal notes>



*)

METHOD xorMaskIsNotEqualTo
VAR_INPUT
	(* current value to check *)
	currentValue	:BYTE;
	(* 2nd operand for bitwise operation *)
	mask			:BYTE;
	(* unexpected result after masking *)
	unexpectedValue	:BYTE;
	(* message if the assertion is false *)
	message			:AssertMessage;
END_VAR
END_METHOD

END_INTERFACE

// ---- Assertor/Assertions/BitNumberAssertions/Dword/interfaces/IDwordAssertions.TcIO
(*

## Short summary
This interface provides assert statements for double words  

.. <legal notes>

legal notes
=================
| SPDX-FileCopyrightText: © 2022 ekvip automation GmbH <info@ekvip.de>
| SPDX-License-Identifier: Apache-2.0
| For details check: Apache-2.0_

.. _Apache-2.0: https://www.apache.org/licenses/LICENSE-2.0

.. </legal notes>



*)

INTERFACE IDwordAssertions EXTENDS __SYSTEM.IQueryInterface

(*

## Short summary
This assertion method checks if the result current value bitwise ``AND`` mask is equal to the expected value

.. <legal notes>

legal notes
=================
| SPDX-FileCopyrightText: © 2022 ekvip automation GmbH <info@ekvip.de>
| SPDX-License-Identifier: Apache-2.0
| For details check: Apache-2.0_

.. _Apache-2.0: https://www.apache.org/licenses/LICENSE-2.0

.. </legal notes>



*)

METHOD andMaskIsEqualTo
VAR_INPUT
	(* current value to check *)
	currentValue	:DWORD;
	(* 2nd operand for bitwise operation *)
	mask			:DWORD;
	(* expected result after masking *)
	expectedValue	:DWORD;
	(* message if the assertion is false *)
	message			:AssertMessage;
END_VAR
END_METHOD

(*

## Short summary
This assertion method checks if the result current value bitwise ``AND`` mask
is not equal to the unexpected value

.. <legal notes>

legal notes
=================
| SPDX-FileCopyrightText: © 2022 ekvip automation GmbH <info@ekvip.de>
| SPDX-License-Identifier: Apache-2.0
| For details check: Apache-2.0_

.. _Apache-2.0: https://www.apache.org/licenses/LICENSE-2.0

.. </legal notes>



*)

METHOD andMaskIsNotEqualTo
VAR_INPUT
	(* current value to check *)
	currentValue	:DWORD;
	(* 2nd operand for bitwise operation *)
	mask			:DWORD;
	(* unexpected result after masking *)
	unexpectedValue	:DWORD;
	(* message if the assertion is false *)
	message			:AssertMessage;
END_VAR
END_METHOD

(*

## Short summary
This assertion method checks if the selected bit of current value
is equal to the expected value

.. <legal notes>

legal notes
=================
| SPDX-FileCopyrightText: © 2022 ekvip automation GmbH <info@ekvip.de>
| SPDX-License-Identifier: Apache-2.0
| For details check: Apache-2.0_

.. _Apache-2.0: https://www.apache.org/licenses/LICENSE-2.0

.. </legal notes>



*)

METHOD bitXIsEqualTo
VAR_INPUT
	(* current value to check *)
	currentValue	:DWORD;
	(* number of bit to check *)
	number			:BitNumberDWord;	
	(* expected value of bit *)
	expectedValue	:BOOL;
	(* message if the assertion is false *)
	message			:AssertMessage;
END_VAR
END_METHOD

(*

## Short summary
This assertion method checks if the selected bit of current value
is not equal to the unexpected value

.. <legal notes>

legal notes
=================
| SPDX-FileCopyrightText: © 2022 ekvip automation GmbH <info@ekvip.de>
| SPDX-License-Identifier: Apache-2.0
| For details check: Apache-2.0_

.. _Apache-2.0: https://www.apache.org/licenses/LICENSE-2.0

.. </legal notes>



*)

METHOD bitXIsNotEqualTo
VAR_INPUT
	(* current value to check *)
	currentValue	:DWORD;
	(* number of bit to check *)
	number			:BitNumberDWord;	
	(* unexpected value of bit *)
	unexpectedValue	:BOOL;
	(* message if the assertion is false *)
	message			:AssertMessage;
END_VAR
END_METHOD

(*

## Short summary
This assertion method checks if the selected bit of current value
is set

.. <legal notes>

legal notes
=================
| SPDX-FileCopyrightText: © 2022 ekvip automation GmbH <info@ekvip.de>
| SPDX-License-Identifier: Apache-2.0
| For details check: Apache-2.0_

.. _Apache-2.0: https://www.apache.org/licenses/LICENSE-2.0

.. </legal notes>



*)

METHOD bitXIsSet
VAR_INPUT
	(* current value to check *)
	currentValue	:DWORD;
	(* number of bit to check *)
	number			:BitNumberDWord;	
	(* message if the assertion is false *)
	message			:AssertMessage;
END_VAR
END_METHOD

(*

## Short summary
This assertion method checks if the selected bit of current value
is unset

.. <legal notes>

legal notes
=================
| SPDX-FileCopyrightText: © 2022 ekvip automation GmbH <info@ekvip.de>
| SPDX-License-Identifier: Apache-2.0
| For details check: Apache-2.0_

.. _Apache-2.0: https://www.apache.org/licenses/LICENSE-2.0

.. </legal notes>



*)

METHOD bitXIsUnset
VAR_INPUT
	(* current value to check *)
	currentValue	:DWORD;
	(* number of bit to check *)
	number			:BitNumberDWord;	
	(* message if the assertion is false *)
	message			:AssertMessage;
END_VAR
END_METHOD

(*

## Short summary
This assertion method checks if the least significant bit of current value
is equal to the expected value

.. <legal notes>

legal notes
=================
| SPDX-FileCopyrightText: © 2022 ekvip automation GmbH <info@ekvip.de>
| SPDX-License-Identifier: Apache-2.0
| For details check: Apache-2.0_

.. _Apache-2.0: https://www.apache.org/licenses/LICENSE-2.0

.. </legal notes>



*)

METHOD lsbIsEqualTo
VAR_INPUT
	(* current value to check *)
	currentValue	:DWORD;
	(* expected value of lsb *)
	expectedValue	:BOOL;
	(* message if the assertion is false *)
	message			:AssertMessage;
END_VAR
END_METHOD

(*

## Short summary
This assertion method checks if the least significant bit of current value
is not equal to the unexpected value

.. <legal notes>

legal notes
=================
| SPDX-FileCopyrightText: © 2022 ekvip automation GmbH <info@ekvip.de>
| SPDX-License-Identifier: Apache-2.0
| For details check: Apache-2.0_

.. _Apache-2.0: https://www.apache.org/licenses/LICENSE-2.0

.. </legal notes>



*)

METHOD lsbIsNotEqualTo
VAR_INPUT
	(* current value to check *)
	currentValue	:DWORD;
	(* unexpected value of lsb *)
	unexpectedValue	:BOOL;
	(* message if the assertion is false *)
	message			:AssertMessage;
END_VAR
END_METHOD

(*

## Short summary
This assertion method checks if the least significant bit of current value
is set

.. <legal notes>

legal notes
=================
| SPDX-FileCopyrightText: © 2022 ekvip automation GmbH <info@ekvip.de>
| SPDX-License-Identifier: Apache-2.0
| For details check: Apache-2.0_

.. _Apache-2.0: https://www.apache.org/licenses/LICENSE-2.0

.. </legal notes>



*)

METHOD lsbIsSet
VAR_INPUT
	(* current value to check *)
	currentValue	:DWORD;
	(* message if the assertion is false *)
	message			:AssertMessage;
END_VAR
END_METHOD

(*

## Short summary
This assertion method checks if the least significant bit of current value
is unset

.. <legal notes>

legal notes
=================
| SPDX-FileCopyrightText: © 2022 ekvip automation GmbH <info@ekvip.de>
| SPDX-License-Identifier: Apache-2.0
| For details check: Apache-2.0_

.. _Apache-2.0: https://www.apache.org/licenses/LICENSE-2.0

.. </legal notes>



*)

METHOD lsbIsUnset
VAR_INPUT
	(* current value to check *)
	currentValue	:DWORD;
	(* message if the assertion is false *)
	message			:AssertMessage;
END_VAR
END_METHOD

(*

## Short summary
This assertion method checks if the most significant bit of current value
is equal to the expected value

.. <legal notes>

legal notes
=================
| SPDX-FileCopyrightText: © 2022 ekvip automation GmbH <info@ekvip.de>
| SPDX-License-Identifier: Apache-2.0
| For details check: Apache-2.0_

.. _Apache-2.0: https://www.apache.org/licenses/LICENSE-2.0

.. </legal notes>



*)

METHOD msbIsEqualTo
VAR_INPUT
	(* current value to check *)
	currentValue	:DWORD;
	(* expected value of msb *)
	expectedValue	:BOOL;
	(* message if the assertion is false *)
	message			:AssertMessage;
END_VAR
END_METHOD

(*

## Short summary
This assertion method checks if the most significant bit of current value
is not equal to the unexpected value

.. <legal notes>

legal notes
=================
| SPDX-FileCopyrightText: © 2022 ekvip automation GmbH <info@ekvip.de>
| SPDX-License-Identifier: Apache-2.0
| For details check: Apache-2.0_

.. _Apache-2.0: https://www.apache.org/licenses/LICENSE-2.0

.. </legal notes>



*)

METHOD msbIsNotEqualTo
VAR_INPUT
	(* current value to check *)
	currentValue	:DWORD;
	(* unexpected value of msb *)
	unexpectedValue	:BOOL;
	(* message if the assertion is false *)
	message			:AssertMessage;
END_VAR
END_METHOD

(*

## Short summary
This assertion method checks if the most significant bit of current value
is set

.. <legal notes>

legal notes
=================
| SPDX-FileCopyrightText: © 2022 ekvip automation GmbH <info@ekvip.de>
| SPDX-License-Identifier: Apache-2.0
| For details check: Apache-2.0_

.. _Apache-2.0: https://www.apache.org/licenses/LICENSE-2.0

.. </legal notes>



*)

METHOD msbIsSet
VAR_INPUT
	(* current value to check *)
	currentValue	:DWORD;
	(* message if the assertion is false *)
	message			:AssertMessage;
END_VAR
END_METHOD

(*

## Short summary
This assertion method checks if the most significant bit of current value
is unset

.. <legal notes>

legal notes
=================
| SPDX-FileCopyrightText: © 2022 ekvip automation GmbH <info@ekvip.de>
| SPDX-License-Identifier: Apache-2.0
| For details check: Apache-2.0_

.. _Apache-2.0: https://www.apache.org/licenses/LICENSE-2.0

.. </legal notes>



*)

METHOD msbIsUnset
VAR_INPUT
	(* current value to check *)
	currentValue	:DWORD;
	(* message if the assertion is false *)
	message			:AssertMessage;
END_VAR
END_METHOD

(*

## Short summary
This assertion method checks if the result current value bitwise ``OR`` mask is equal to the expected value

.. <legal notes>

legal notes
=================
| SPDX-FileCopyrightText: © 2022 ekvip automation GmbH <info@ekvip.de>
| SPDX-License-Identifier: Apache-2.0
| For details check: Apache-2.0_

.. _Apache-2.0: https://www.apache.org/licenses/LICENSE-2.0

.. </legal notes>



*)

METHOD orMaskIsEqualTo
VAR_INPUT
	(* current value to check *)
	currentValue	:DWORD;
	(* 2nd operand for bitwise operation *)
	mask			:DWORD;
	(* expected result after masking *)
	expectedValue	:DWORD;
	(* message if the assertion is false *)
	message			:AssertMessage;
END_VAR
END_METHOD

(*

## Short summary
This assertion method checks if the result current value bitwise ``OR`` mask 
is not equal to the unexpected value

.. <legal notes>

legal notes
=================
| SPDX-FileCopyrightText: © 2022 ekvip automation GmbH <info@ekvip.de>
| SPDX-License-Identifier: Apache-2.0
| For details check: Apache-2.0_

.. _Apache-2.0: https://www.apache.org/licenses/LICENSE-2.0

.. </legal notes>



*)

METHOD orMaskIsNotEqualTo
VAR_INPUT
	(* current value to check *)
	currentValue	:DWORD;
	(* 2nd operand for bitwise operation *)
	mask			:DWORD;
	(* unexpected result after masking *)
	unexpectedValue	:DWORD;
	(* message if the assertion is false *)
	message			:AssertMessage;
END_VAR
END_METHOD

(*

## Short summary
This assertion method checks if the current value is equal to the expected value

.. <legal notes>

legal notes
=================
| SPDX-FileCopyrightText: © 2022 ekvip automation GmbH <info@ekvip.de>
| SPDX-License-Identifier: Apache-2.0
| For details check: Apache-2.0_

.. _Apache-2.0: https://www.apache.org/licenses/LICENSE-2.0

.. </legal notes>



*)

METHOD valueIsEqualTo
VAR_INPUT
	(* current value to check *)
	currentValue	:DWORD;
	(* expected value to compare *)
	expectedValue	:DWORD;
	(* message if the assertion is false *)
	message			:AssertMessage;
END_VAR
END_METHOD

(*

## Short summary
This assertion method checks if the current value is greater than the less value

.. <legal notes>

legal notes
=================
| SPDX-FileCopyrightText: © 2022 ekvip automation GmbH <info@ekvip.de>
| SPDX-License-Identifier: Apache-2.0
| For details check: Apache-2.0_

.. _Apache-2.0: https://www.apache.org/licenses/LICENSE-2.0

.. </legal notes>



*)

METHOD valueIsGreaterThan
VAR_INPUT
	(* current value to check *)
	currentValue	:DWORD;
	(* less than lower limit *)
	lessValue		:DWORD;
	(* message if the assertion is false *)
	message			:AssertMessage;
END_VAR
END_METHOD

(*

## Short summary
This assertion method checks if the current value is inside a limit

**Attention:** 
	limits are included: ``valueIsInRangeOf(3, 3, 3)`` is a true assertion

.. <legal notes>

legal notes
=================
| SPDX-FileCopyrightText: © 2022 ekvip automation GmbH <info@ekvip.de>
| SPDX-License-Identifier: Apache-2.0
| For details check: Apache-2.0_

.. _Apache-2.0: https://www.apache.org/licenses/LICENSE-2.0

.. </legal notes>



*)

METHOD valueIsInRangeOf
VAR_INPUT
	(* lower limit for the current value *)
	lowerLimit		:DWORD;
	(* current value to check *)
	currentValue	:DWORD;
	(* upper limit for the current value *)
	upperLimit		:DWORD;
	(* message if the assertion is false *)
	message			:AssertMessage;
END_VAR
END_METHOD

(*

## Short summary
This assertion method checks if the current value is less than the greater value

.. <legal notes>

legal notes
=================
| SPDX-FileCopyrightText: © 2022 ekvip automation GmbH <info@ekvip.de>
| SPDX-License-Identifier: Apache-2.0
| For details check: Apache-2.0_

.. _Apache-2.0: https://www.apache.org/licenses/LICENSE-2.0

.. </legal notes>



*)

METHOD valueIsLessThan
VAR_INPUT
	(* current value to check *)
	currentValue	:DWORD;
	(* greater than upper limit *)
	greaterValue	:DWORD;
	(* message if the assertion is false *)
	message			:AssertMessage;
END_VAR
END_METHOD

(*

## Short summary
This assertion method checks if the current value is less than or equal to the maximum value

.. <legal notes>

legal notes
=================
| SPDX-FileCopyrightText: © 2022 ekvip automation GmbH <info@ekvip.de>
| SPDX-License-Identifier: Apache-2.0
| For details check: Apache-2.0_

.. _Apache-2.0: https://www.apache.org/licenses/LICENSE-2.0

.. </legal notes>



*)

METHOD valueIsMax
VAR_INPUT
	(* current value to check *)
	currentValue	:DWORD;
	(* upper limit for the current value *)
	maximumValue	:DWORD;
	(* message if the assertion is false *)
	message			:AssertMessage;
END_VAR
END_METHOD

(*

## Short summary
This assertion method checks if the current value is greater than or equal to the minimum value

.. <legal notes>

legal notes
=================
| SPDX-FileCopyrightText: © 2022 ekvip automation GmbH <info@ekvip.de>
| SPDX-License-Identifier: Apache-2.0
| For details check: Apache-2.0_

.. _Apache-2.0: https://www.apache.org/licenses/LICENSE-2.0

.. </legal notes>



*)

METHOD valueIsMin
VAR_INPUT
	(* current value to check *)
	currentValue	:DWORD;
	(* lower limit for the current value *)
	minimumValue	:DWORD;
	(* message if the assertion is false *)
	message			:AssertMessage;
END_VAR
END_METHOD

(*

## Short summary
This assertion method checks if the current value is not equal to the unexpected value

.. <legal notes>

legal notes
=================
| SPDX-FileCopyrightText: © 2022 ekvip automation GmbH <info@ekvip.de>
| SPDX-License-Identifier: Apache-2.0
| For details check: Apache-2.0_

.. _Apache-2.0: https://www.apache.org/licenses/LICENSE-2.0

.. </legal notes>



*)

METHOD valueIsNotEqualTo
VAR_INPUT
	(* current value to check *)
	currentValue	:DWORD;
	(* unexpected value to compare *)
	unexpectedValue	:DWORD;
	(* message if the assertion is false *)
	message			:AssertMessage;
END_VAR
END_METHOD

(*

## Short summary
This assertion method checks if the result current value bitwise ``XOR`` mask is equal to the expected value

.. <legal notes>

legal notes
=================
| SPDX-FileCopyrightText: © 2022 ekvip automation GmbH <info@ekvip.de>
| SPDX-License-Identifier: Apache-2.0
| For details check: Apache-2.0_

.. _Apache-2.0: https://www.apache.org/licenses/LICENSE-2.0

.. </legal notes>



*)

METHOD xorMaskIsEqualTo
VAR_INPUT
	(* current value to check *)
	currentValue	:DWORD;
	(* 2nd operand for bitwise operation *)
	mask			:DWORD;
	(* expected result after masking *)
	expectedValue	:DWORD;
	(* message if the assertion is false *)
	message			:AssertMessage;
END_VAR
END_METHOD

(*

## Short summary
This assertion method checks if the result current value bitwise ``XOR`` mask 
is not equal to the unexpected value

.. <legal notes>

legal notes
=================
| SPDX-FileCopyrightText: © 2022 ekvip automation GmbH <info@ekvip.de>
| SPDX-License-Identifier: Apache-2.0
| For details check: Apache-2.0_

.. _Apache-2.0: https://www.apache.org/licenses/LICENSE-2.0

.. </legal notes>



*)

METHOD xorMaskIsNotEqualTo
VAR_INPUT
	(* current value to check *)
	currentValue	:DWORD;
	(* 2nd operand for bitwise operation *)
	mask			:DWORD;
	(* unexpected result after masking *)
	unexpectedValue	:DWORD;
	(* message if the assertion is false *)
	message			:AssertMessage;
END_VAR
END_METHOD

END_INTERFACE

// ---- Assertor/Assertions/BitNumberAssertions/interfaces/IBitNumberAssertions.TcIO
(*

## Short summary

This interface provides assert statements for bit numbers:
For ``BYTE`` use `IBitNumberAssertions.short`
For ``WORD`` use `IBitNumberAssertions.simple`
For ``DWORD`` use `IBitNumberAssertions.double`
For ``LWORD`` use `IBitNumberAssertions.long`
For ``__XWORD`` use `IBitNumberAssertions.x`

.. <legal notes>

legal notes
=================
| SPDX-FileCopyrightText: © 2022 ekvip automation GmbH <info@ekvip.de>
| SPDX-License-Identifier: Apache-2.0
| For details check: Apache-2.0_

.. _Apache-2.0: https://www.apache.org/licenses/LICENSE-2.0

.. </legal notes>

properties
==================

*)

INTERFACE IBitNumberAssertions EXTENDS __SYSTEM.IQueryInterface

(*

## Short summary
Returns the interface `IDwordAssertions`
with assert statements for double words ``DWORD`` 

.. <legal notes>

legal notes
=================
| SPDX-FileCopyrightText: © 2022 ekvip automation GmbH <info@ekvip.de>
| SPDX-License-Identifier: Apache-2.0
| For details check: Apache-2.0_

.. _Apache-2.0: https://www.apache.org/licenses/LICENSE-2.0

.. </legal notes>

*)

PROPERTY double :IDwordAssertions
GET
END_GET
END_PROPERTY

(*

## Short summary
Returns the interface `ILwordAssertions`
with assert statements for long words ``LWORD`` 

.. <legal notes>

legal notes
=================
| SPDX-FileCopyrightText: © 2022 ekvip automation GmbH <info@ekvip.de>
| SPDX-License-Identifier: Apache-2.0
| For details check: Apache-2.0_

.. _Apache-2.0: https://www.apache.org/licenses/LICENSE-2.0

.. </legal notes>

*)

PROPERTY long :ILwordAssertions
GET
END_GET
END_PROPERTY

(*

## Short summary
Returns the interface `IByteAssertions`
with assert statements for bytes

.. <legal notes>

legal notes
=================
| SPDX-FileCopyrightText: © 2022 ekvip automation GmbH <info@ekvip.de>
| SPDX-License-Identifier: Apache-2.0
| For details check: Apache-2.0_

.. _Apache-2.0: https://www.apache.org/licenses/LICENSE-2.0

.. </legal notes>

*)

PROPERTY short :IByteAssertions
GET
END_GET
END_PROPERTY

(*

## Short summary
Returns the interface `IWordAssertions`
with assert statements for words 

.. <legal notes>

legal notes
=================
| SPDX-FileCopyrightText: © 2022 ekvip automation GmbH <info@ekvip.de>
| SPDX-License-Identifier: Apache-2.0
| For details check: Apache-2.0_

.. _Apache-2.0: https://www.apache.org/licenses/LICENSE-2.0

.. </legal notes>

*)

PROPERTY simple :IWordAssertions
GET
END_GET
END_PROPERTY

(*

## Short summary
Returns the interface `IXwordAssertions`
with assert statements for register length words ``__XWORD``

.. <legal notes>

legal notes
=================
| SPDX-FileCopyrightText: © 2022 ekvip automation GmbH <info@ekvip.de>
| SPDX-License-Identifier: Apache-2.0
| For details check: Apache-2.0_

.. _Apache-2.0: https://www.apache.org/licenses/LICENSE-2.0

.. </legal notes>

*)

PROPERTY x :IXwordAssertions
GET
END_GET
END_PROPERTY

END_INTERFACE

// ---- Assertor/Assertions/BitNumberAssertions/Lword/interfaces/ILwordAssertions.TcIO
(*

## Short summary
This interface provides assert statements for long words  

.. <legal notes>

legal notes
=================
| SPDX-FileCopyrightText: © 2022 ekvip automation GmbH <info@ekvip.de>
| SPDX-License-Identifier: Apache-2.0
| For details check: Apache-2.0_

.. _Apache-2.0: https://www.apache.org/licenses/LICENSE-2.0

.. </legal notes>



*)

INTERFACE ILwordAssertions EXTENDS __SYSTEM.IQueryInterface

(*

## Short summary
This assertion method checks if the result current value bitwise ``AND`` mask is equal to the expected value

.. <legal notes>

legal notes
=================
| SPDX-FileCopyrightText: © 2022 ekvip automation GmbH <info@ekvip.de>
| SPDX-License-Identifier: Apache-2.0
| For details check: Apache-2.0_

.. _Apache-2.0: https://www.apache.org/licenses/LICENSE-2.0

.. </legal notes>



*)

METHOD andMaskIsEqualTo
VAR_INPUT
	(* current value to check *)
	currentValue	:LWORD;
	(* 2nd operand for bitwise operation *)
	mask			:LWORD;
	(* expected result after masking *)
	expectedValue	:LWORD;
	(* message if the assertion is false *)
	message			:AssertMessage;
END_VAR
END_METHOD

(*

## Short summary
This assertion method checks if the result current value bitwise ``AND`` mask
is not equal to the unexpected value

.. <legal notes>

legal notes
=================
| SPDX-FileCopyrightText: © 2022 ekvip automation GmbH <info@ekvip.de>
| SPDX-License-Identifier: Apache-2.0
| For details check: Apache-2.0_

.. _Apache-2.0: https://www.apache.org/licenses/LICENSE-2.0

.. </legal notes>



*)

METHOD andMaskIsNotEqualTo
VAR_INPUT
	(* current value to check *)
	currentValue	:LWORD;
	(* 2nd operand for bitwise operation *)
	mask			:LWORD;
	(* unexpected result after masking *)
	unexpectedValue	:LWORD;
	(* message if the assertion is false *)
	message			:AssertMessage;
END_VAR
END_METHOD

(*

## Short summary
This assertion method checks if the selected bit of current value
is equal to the expected value

.. <legal notes>

legal notes
=================
| SPDX-FileCopyrightText: © 2022 ekvip automation GmbH <info@ekvip.de>
| SPDX-License-Identifier: Apache-2.0
| For details check: Apache-2.0_

.. _Apache-2.0: https://www.apache.org/licenses/LICENSE-2.0

.. </legal notes>



*)

METHOD bitXIsEqualTo
VAR_INPUT
	(* current value to check *)
	currentValue	:LWORD;
	(* number of bit to check *)
	number			:BitNumberLWord;	
	(* expected value of bit *)
	expectedValue	:BOOL;
	(* message if the assertion is false *)
	message			:AssertMessage;
END_VAR
END_METHOD

(*

## Short summary
This assertion method checks if the selected bit of current value
is not equal to the unexpected value

.. <legal notes>

legal notes
=================
| SPDX-FileCopyrightText: © 2022 ekvip automation GmbH <info@ekvip.de>
| SPDX-License-Identifier: Apache-2.0
| For details check: Apache-2.0_

.. _Apache-2.0: https://www.apache.org/licenses/LICENSE-2.0

.. </legal notes>



*)

METHOD bitXIsNotEqualTo
VAR_INPUT
	(* current value to check *)
	currentValue	:LWORD;
	(* number of bit to check *)
	number			:BitNumberLWord;	
	(* unexpected value of bit *)
	unexpectedValue	:BOOL;
	(* message if the assertion is false *)
	message			:AssertMessage;
END_VAR
END_METHOD

(*

## Short summary
This assertion method checks if the selected bit of current value
is set

.. <legal notes>

legal notes
=================
| SPDX-FileCopyrightText: © 2022 ekvip automation GmbH <info@ekvip.de>
| SPDX-License-Identifier: Apache-2.0
| For details check: Apache-2.0_

.. _Apache-2.0: https://www.apache.org/licenses/LICENSE-2.0

.. </legal notes>



*)

METHOD bitXIsSet
VAR_INPUT
	(* current value to check *)
	currentValue	:LWORD;
	(* number of bit to check *)
	number			:BitNumberLWord;	
	(* message if the assertion is false *)
	message			:AssertMessage;
END_VAR
END_METHOD

(*

## Short summary
This assertion method checks if the selected bit of current value
is unset

.. <legal notes>

legal notes
=================
| SPDX-FileCopyrightText: © 2022 ekvip automation GmbH <info@ekvip.de>
| SPDX-License-Identifier: Apache-2.0
| For details check: Apache-2.0_

.. _Apache-2.0: https://www.apache.org/licenses/LICENSE-2.0

.. </legal notes>



*)

METHOD bitXIsUnset
VAR_INPUT
	(* current value to check *)
	currentValue	:LWORD;
	(* number of bit to check *)
	number			:BitNumberLWord;	
	(* message if the assertion is false *)
	message			:AssertMessage;
END_VAR
END_METHOD

(*

## Short summary
This assertion method checks if the least significant bit of current value
is equal to the expected value

.. <legal notes>

legal notes
=================
| SPDX-FileCopyrightText: © 2022 ekvip automation GmbH <info@ekvip.de>
| SPDX-License-Identifier: Apache-2.0
| For details check: Apache-2.0_

.. _Apache-2.0: https://www.apache.org/licenses/LICENSE-2.0

.. </legal notes>



*)

METHOD lsbIsEqualTo
VAR_INPUT
	(* current value to check *)
	currentValue	:LWORD;
	(* expected value of lsb *)
	expectedValue	:BOOL;
	(* message if the assertion is false *)
	message			:AssertMessage;
END_VAR
END_METHOD

(*

## Short summary
This assertion method checks if the least significant bit of current value
is not equal to the unexpected value

.. <legal notes>

legal notes
=================
| SPDX-FileCopyrightText: © 2022 ekvip automation GmbH <info@ekvip.de>
| SPDX-License-Identifier: Apache-2.0
| For details check: Apache-2.0_

.. _Apache-2.0: https://www.apache.org/licenses/LICENSE-2.0

.. </legal notes>



*)

METHOD lsbIsNotEqualTo
VAR_INPUT
	(* current value to check *)
	currentValue	:LWORD;
	(* unexpected value of lsb *)
	unexpectedValue	:BOOL;
	(* message if the assertion is false *)
	message			:AssertMessage;
END_VAR
END_METHOD

(*

## Short summary
This assertion method checks if the least significant bit of current value
is set

.. <legal notes>

legal notes
=================
| SPDX-FileCopyrightText: © 2022 ekvip automation GmbH <info@ekvip.de>
| SPDX-License-Identifier: Apache-2.0
| For details check: Apache-2.0_

.. _Apache-2.0: https://www.apache.org/licenses/LICENSE-2.0

.. </legal notes>



*)

METHOD lsbIsSet
VAR_INPUT
	(* current value to check *)
	currentValue	:LWORD;
	(* message if the assertion is false *)
	message			:AssertMessage;
END_VAR
END_METHOD

(*

## Short summary
This assertion method checks if the least significant bit of current value
is unset

.. <legal notes>

legal notes
=================
| SPDX-FileCopyrightText: © 2022 ekvip automation GmbH <info@ekvip.de>
| SPDX-License-Identifier: Apache-2.0
| For details check: Apache-2.0_

.. _Apache-2.0: https://www.apache.org/licenses/LICENSE-2.0

.. </legal notes>



*)

METHOD lsbIsUnset
VAR_INPUT
	(* current value to check *)
	currentValue	:LWORD;
	(* message if the assertion is false *)
	message			:AssertMessage;
END_VAR
END_METHOD

(*

## Short summary
This assertion method checks if the most significant bit of current value
is equal to the expected value

.. <legal notes>

legal notes
=================
| SPDX-FileCopyrightText: © 2022 ekvip automation GmbH <info@ekvip.de>
| SPDX-License-Identifier: Apache-2.0
| For details check: Apache-2.0_

.. _Apache-2.0: https://www.apache.org/licenses/LICENSE-2.0

.. </legal notes>



*)

METHOD msbIsEqualTo
VAR_INPUT
	(* current value to check *)
	currentValue	:LWORD;
	(* expected value of msb *)
	expectedValue	:BOOL;
	(* message if the assertion is false *)
	message			:AssertMessage;
END_VAR
END_METHOD

(*

## Short summary
This assertion method checks if the most significant bit of current value
is not equal to the unexpected value

.. <legal notes>

legal notes
=================
| SPDX-FileCopyrightText: © 2022 ekvip automation GmbH <info@ekvip.de>
| SPDX-License-Identifier: Apache-2.0
| For details check: Apache-2.0_

.. _Apache-2.0: https://www.apache.org/licenses/LICENSE-2.0

.. </legal notes>



*)

METHOD msbIsNotEqualTo
VAR_INPUT
	(* current value to check *)
	currentValue	:LWORD;
	(* unexpected value of msb *)
	unexpectedValue	:BOOL;
	(* message if the assertion is false *)
	message			:AssertMessage;
END_VAR
END_METHOD

(*

## Short summary
This assertion method checks if the most significant bit of current value
is set

.. <legal notes>

legal notes
=================
| SPDX-FileCopyrightText: © 2022 ekvip automation GmbH <info@ekvip.de>
| SPDX-License-Identifier: Apache-2.0
| For details check: Apache-2.0_

.. _Apache-2.0: https://www.apache.org/licenses/LICENSE-2.0

.. </legal notes>



*)

METHOD msbIsSet
VAR_INPUT
	(* current value to check *)
	currentValue	:LWORD;
	(* message if the assertion is false *)
	message			:AssertMessage;
END_VAR
END_METHOD

(*

## Short summary
This assertion method checks if the most significant bit of current value
is unset

.. <legal notes>

legal notes
=================
| SPDX-FileCopyrightText: © 2022 ekvip automation GmbH <info@ekvip.de>
| SPDX-License-Identifier: Apache-2.0
| For details check: Apache-2.0_

.. _Apache-2.0: https://www.apache.org/licenses/LICENSE-2.0

.. </legal notes>



*)

METHOD msbIsUnset
VAR_INPUT
	(* current value to check *)
	currentValue	:LWORD;
	(* message if the assertion is false *)
	message			:AssertMessage;
END_VAR
END_METHOD

(*

## Short summary
This assertion method checks if the result current value bitwise ``OR`` mask is equal to the expected value

.. <legal notes>

legal notes
=================
| SPDX-FileCopyrightText: © 2022 ekvip automation GmbH <info@ekvip.de>
| SPDX-License-Identifier: Apache-2.0
| For details check: Apache-2.0_

.. _Apache-2.0: https://www.apache.org/licenses/LICENSE-2.0

.. </legal notes>



*)

METHOD orMaskIsEqualTo
VAR_INPUT
	(* current value to check *)
	currentValue	:LWORD;
	(* 2nd operand for bitwise operation *)
	mask			:LWORD;
	(* expected result after masking *)
	expectedValue	:LWORD;
	(* message if the assertion is false *)
	message			:AssertMessage;
END_VAR
END_METHOD

(*

## Short summary
This assertion method checks if the result current value bitwise ``OR`` mask 
is not equal to the unexpected value

.. <legal notes>

legal notes
=================
| SPDX-FileCopyrightText: © 2022 ekvip automation GmbH <info@ekvip.de>
| SPDX-License-Identifier: Apache-2.0
| For details check: Apache-2.0_

.. _Apache-2.0: https://www.apache.org/licenses/LICENSE-2.0

.. </legal notes>



*)

METHOD orMaskIsNotEqualTo
VAR_INPUT
	(* current value to check *)
	currentValue	:LWORD;
	(* 2nd operand for bitwise operation *)
	mask			:LWORD;
	(* unexpected result after masking *)
	unexpectedValue	:LWORD;
	(* message if the assertion is false *)
	message			:AssertMessage;
END_VAR
END_METHOD

(*

## Short summary
This assertion method checks if the current value is equal to the expected value

.. <legal notes>

legal notes
=================
| SPDX-FileCopyrightText: © 2022 ekvip automation GmbH <info@ekvip.de>
| SPDX-License-Identifier: Apache-2.0
| For details check: Apache-2.0_

.. _Apache-2.0: https://www.apache.org/licenses/LICENSE-2.0

.. </legal notes>



*)

METHOD valueIsEqualTo
VAR_INPUT
	(* current value to check *)
	currentValue	:LWORD;
	(* expected value to compare *)
	expectedValue	:LWORD;
	(* message if the assertion is false *)
	message			:AssertMessage;
END_VAR
END_METHOD

(*

## Short summary
This assertion method checks if the current value is greater than the less value

.. <legal notes>

legal notes
=================
| SPDX-FileCopyrightText: © 2022 ekvip automation GmbH <info@ekvip.de>
| SPDX-License-Identifier: Apache-2.0
| For details check: Apache-2.0_

.. _Apache-2.0: https://www.apache.org/licenses/LICENSE-2.0

.. </legal notes>



*)

METHOD valueIsGreaterThan
VAR_INPUT
	(* current value to check *)
	currentValue	:LWORD;
	(* less than lower limit *)
	lessValue		:LWORD;
	(* message if the assertion is false *)
	message			:AssertMessage;
END_VAR
END_METHOD

(*

## Short summary
This assertion method checks if the current value is inside a limit

**Attention:** 
	limits are included: ``valueIsInRangeOf(3, 3, 3)`` is a true assertion

.. <legal notes>

legal notes
=================
| SPDX-FileCopyrightText: © 2022 ekvip automation GmbH <info@ekvip.de>
| SPDX-License-Identifier: Apache-2.0
| For details check: Apache-2.0_

.. _Apache-2.0: https://www.apache.org/licenses/LICENSE-2.0

.. </legal notes>



*)

METHOD valueIsInRangeOf
VAR_INPUT
	(* lower limit for the current value *)
	lowerLimit		:LWORD;
	(* current value to check *)
	currentValue	:LWORD;
	(* upper limit for the current value *)
	upperLimit		:LWORD;
	(* message if the assertion is false *)
	message			:AssertMessage;
END_VAR
END_METHOD

(*

## Short summary
This assertion method checks if the current value is less than the greater value

.. <legal notes>

legal notes
=================
| SPDX-FileCopyrightText: © 2022 ekvip automation GmbH <info@ekvip.de>
| SPDX-License-Identifier: Apache-2.0
| For details check: Apache-2.0_

.. _Apache-2.0: https://www.apache.org/licenses/LICENSE-2.0

.. </legal notes>



*)

METHOD valueIsLessThan
VAR_INPUT
	(* current value to check *)
	currentValue	:LWORD;
	(* greater than upper limit *)
	greaterValue	:LWORD;
	(* message if the assertion is false *)
	message			:AssertMessage;
END_VAR
END_METHOD

(*

## Short summary
This assertion method checks if the current value is less than or equal to the maximum value

.. <legal notes>

legal notes
=================
| SPDX-FileCopyrightText: © 2022 ekvip automation GmbH <info@ekvip.de>
| SPDX-License-Identifier: Apache-2.0
| For details check: Apache-2.0_

.. _Apache-2.0: https://www.apache.org/licenses/LICENSE-2.0

.. </legal notes>



*)

METHOD valueIsMax
VAR_INPUT
	(* current value to check *)
	currentValue	:LWORD;
	(* upper limit for the current value *)
	maximumValue	:LWORD;
	(* message if the assertion is false *)
	message			:AssertMessage;
END_VAR
END_METHOD

(*

## Short summary
This assertion method checks if the current value is greater than or equal to the minimum value

.. <legal notes>

legal notes
=================
| SPDX-FileCopyrightText: © 2022 ekvip automation GmbH <info@ekvip.de>
| SPDX-License-Identifier: Apache-2.0
| For details check: Apache-2.0_

.. _Apache-2.0: https://www.apache.org/licenses/LICENSE-2.0

.. </legal notes>



*)

METHOD valueIsMin
VAR_INPUT
	(* current value to check *)
	currentValue	:LWORD;
	(* lower limit for the current value *)
	minimumValue	:LWORD;
	(* message if the assertion is false *)
	message			:AssertMessage;
END_VAR
END_METHOD

(*

## Short summary
This assertion method checks if the current value is not equal to the unexpected value

.. <legal notes>

legal notes
=================
| SPDX-FileCopyrightText: © 2022 ekvip automation GmbH <info@ekvip.de>
| SPDX-License-Identifier: Apache-2.0
| For details check: Apache-2.0_

.. _Apache-2.0: https://www.apache.org/licenses/LICENSE-2.0

.. </legal notes>



*)

METHOD valueIsNotEqualTo
VAR_INPUT
	(* current value to check *)
	currentValue	:LWORD;
	(* unexpected value to compare *)
	unexpectedValue	:LWORD;
	(* message if the assertion is false *)
	message			:AssertMessage;
END_VAR
END_METHOD

(*

## Short summary
This assertion method checks if the result current value bitwise ``XOR`` mask is equal to the expected value

.. <legal notes>

legal notes
=================
| SPDX-FileCopyrightText: © 2022 ekvip automation GmbH <info@ekvip.de>
| SPDX-License-Identifier: Apache-2.0
| For details check: Apache-2.0_

.. _Apache-2.0: https://www.apache.org/licenses/LICENSE-2.0

.. </legal notes>



*)

METHOD xorMaskIsEqualTo
VAR_INPUT
	(* current value to check *)
	currentValue	:LWORD;
	(* 2nd operand for bitwise operation *)
	mask			:LWORD;
	(* expected result after masking *)
	expectedValue	:LWORD;
	(* message if the assertion is false *)
	message			:AssertMessage;
END_VAR
END_METHOD

(*

## Short summary
This assertion method checks if the result current value bitwise ``XOR`` mask 
is not equal to the unexpected value

.. <legal notes>

legal notes
=================
| SPDX-FileCopyrightText: © 2022 ekvip automation GmbH <info@ekvip.de>
| SPDX-License-Identifier: Apache-2.0
| For details check: Apache-2.0_

.. _Apache-2.0: https://www.apache.org/licenses/LICENSE-2.0

.. </legal notes>



*)

METHOD xorMaskIsNotEqualTo
VAR_INPUT
	(* current value to check *)
	currentValue	:LWORD;
	(* 2nd operand for bitwise operation *)
	mask			:LWORD;
	(* unexpected result after masking *)
	unexpectedValue	:LWORD;
	(* message if the assertion is false *)
	message			:AssertMessage;
END_VAR
END_METHOD

END_INTERFACE

// ---- Assertor/Assertions/BitNumberAssertions/Word/interfaces/IWordAssertions.TcIO
(*

## Short summary
This interface provides assert statements for words  

.. <legal notes>

legal notes
=================
| SPDX-FileCopyrightText: © 2022 ekvip automation GmbH <info@ekvip.de>
| SPDX-License-Identifier: Apache-2.0
| For details check: Apache-2.0_

.. _Apache-2.0: https://www.apache.org/licenses/LICENSE-2.0

.. </legal notes>



*)

INTERFACE IWordAssertions EXTENDS __SYSTEM.IQueryInterface

(*

## Short summary
This assertion method checks if the result current value bitwise ``AND`` mask is equal to the expected value

.. <legal notes>

legal notes
=================
| SPDX-FileCopyrightText: © 2022 ekvip automation GmbH <info@ekvip.de>
| SPDX-License-Identifier: Apache-2.0
| For details check: Apache-2.0_

.. _Apache-2.0: https://www.apache.org/licenses/LICENSE-2.0

.. </legal notes>



*)

METHOD andMaskIsEqualTo
VAR_INPUT
	(* current value to check *)
	currentValue	:WORD;
	(* 2nd operand for bitwise operation *)
	mask			:WORD;
	(* expected result after masking *)
	expectedValue	:WORD;
	(* message if the assertion is false *)
	message			:AssertMessage;
END_VAR
END_METHOD

(*

## Short summary
This assertion method checks if the result current value bitwise ``AND`` mask
is not equal to the unexpected value

.. <legal notes>

legal notes
=================
| SPDX-FileCopyrightText: © 2022 ekvip automation GmbH <info@ekvip.de>
| SPDX-License-Identifier: Apache-2.0
| For details check: Apache-2.0_

.. _Apache-2.0: https://www.apache.org/licenses/LICENSE-2.0

.. </legal notes>



*)

METHOD andMaskIsNotEqualTo
VAR_INPUT
	(* current value to check *)
	currentValue	:WORD;
	(* 2nd operand for bitwise operation *)
	mask			:WORD;
	(* unexpected result after masking *)
	unexpectedValue	:WORD;
	(* message if the assertion is false *)
	message			:AssertMessage;
END_VAR
END_METHOD

(*

## Short summary
This assertion method checks if the selected bit of current value
is equal to the expected value

.. <legal notes>

legal notes
=================
| SPDX-FileCopyrightText: © 2022 ekvip automation GmbH <info@ekvip.de>
| SPDX-License-Identifier: Apache-2.0
| For details check: Apache-2.0_

.. _Apache-2.0: https://www.apache.org/licenses/LICENSE-2.0

.. </legal notes>



*)

METHOD bitXIsEqualTo
VAR_INPUT
	(* current value to check *)
	currentValue	:WORD;
	(* number of bit to check *)
	number			:BitNumberWord;	
	(* expected value of bit *)
	expectedValue	:BOOL;
	(* message if the assertion is false *)
	message			:AssertMessage;
END_VAR
END_METHOD

(*

## Short summary
This assertion method checks if the selected bit of current value
is not equal to the unexpected value

.. <legal notes>

legal notes
=================
| SPDX-FileCopyrightText: © 2022 ekvip automation GmbH <info@ekvip.de>
| SPDX-License-Identifier: Apache-2.0
| For details check: Apache-2.0_

.. _Apache-2.0: https://www.apache.org/licenses/LICENSE-2.0

.. </legal notes>



*)

METHOD bitXIsNotEqualTo
VAR_INPUT
	(* current value to check *)
	currentValue	:WORD;
	(* number of bit to check *)
	number			:BitNumberWord;	
	(* unexpected value of bit *)
	unexpectedValue	:BOOL;
	(* message if the assertion is false *)
	message			:AssertMessage;
END_VAR
END_METHOD

(*

## Short summary
This assertion method checks if the selected bit of current value
is set

.. <legal notes>

legal notes
=================
| SPDX-FileCopyrightText: © 2022 ekvip automation GmbH <info@ekvip.de>
| SPDX-License-Identifier: Apache-2.0
| For details check: Apache-2.0_

.. _Apache-2.0: https://www.apache.org/licenses/LICENSE-2.0

.. </legal notes>



*)

METHOD bitXIsSet
VAR_INPUT
	(* current value to check *)
	currentValue	:WORD;
	(* number of bit to check *)
	number			:BitNumberWord;	
	(* message if the assertion is false *)
	message			:AssertMessage;
END_VAR
END_METHOD

(*

## Short summary
This assertion method checks if the selected bit of current value
is unset

.. <legal notes>

legal notes
=================
| SPDX-FileCopyrightText: © 2022 ekvip automation GmbH <info@ekvip.de>
| SPDX-License-Identifier: Apache-2.0
| For details check: Apache-2.0_

.. _Apache-2.0: https://www.apache.org/licenses/LICENSE-2.0

.. </legal notes>



*)

METHOD bitXIsUnset
VAR_INPUT
	(* current value to check *)
	currentValue	:WORD;
	(* number of bit to check *)
	number			:BitNumberWord;	
	(* message if the assertion is false *)
	message			:AssertMessage;
END_VAR
END_METHOD

(*

## Short summary
This assertion method checks if the least significant bit of current value
is equal to the expected value

.. <legal notes>

legal notes
=================
| SPDX-FileCopyrightText: © 2022 ekvip automation GmbH <info@ekvip.de>
| SPDX-License-Identifier: Apache-2.0
| For details check: Apache-2.0_

.. _Apache-2.0: https://www.apache.org/licenses/LICENSE-2.0

.. </legal notes>



*)

METHOD lsbIsEqualTo
VAR_INPUT
	(* current value to check *)
	currentValue	:WORD;
	(* expected value of lsb *)
	expectedValue	:BOOL;
	(* message if the assertion is false *)
	message			:AssertMessage;
END_VAR
END_METHOD

(*

## Short summary
This assertion method checks if the least significant bit of current value
is not equal to the unexpected value

.. <legal notes>

legal notes
=================
| SPDX-FileCopyrightText: © 2022 ekvip automation GmbH <info@ekvip.de>
| SPDX-License-Identifier: Apache-2.0
| For details check: Apache-2.0_

.. _Apache-2.0: https://www.apache.org/licenses/LICENSE-2.0

.. </legal notes>



*)

METHOD lsbIsNotEqualTo
VAR_INPUT
	(* current value to check *)
	currentValue	:WORD;
	(* unexpected value of lsb *)
	unexpectedValue	:BOOL;
	(* message if the assertion is false *)
	message			:AssertMessage;
END_VAR
END_METHOD

(*

## Short summary
This assertion method checks if the least significant bit of current value
is set

.. <legal notes>

legal notes
=================
| SPDX-FileCopyrightText: © 2022 ekvip automation GmbH <info@ekvip.de>
| SPDX-License-Identifier: Apache-2.0
| For details check: Apache-2.0_

.. _Apache-2.0: https://www.apache.org/licenses/LICENSE-2.0

.. </legal notes>



*)

METHOD lsbIsSet
VAR_INPUT
	(* current value to check *)
	currentValue	:WORD;
	(* message if the assertion is false *)
	message			:AssertMessage;
END_VAR
END_METHOD

(*

## Short summary
This assertion method checks if the least significant bit of current value
is unset

.. <legal notes>

legal notes
=================
| SPDX-FileCopyrightText: © 2022 ekvip automation GmbH <info@ekvip.de>
| SPDX-License-Identifier: Apache-2.0
| For details check: Apache-2.0_

.. _Apache-2.0: https://www.apache.org/licenses/LICENSE-2.0

.. </legal notes>



*)

METHOD lsbIsUnset
VAR_INPUT
	(* current value to check *)
	currentValue	:WORD;
	(* message if the assertion is false *)
	message			:AssertMessage;
END_VAR
END_METHOD

(*

## Short summary
This assertion method checks if the most significant bit of current value
is equal to the expected value

.. <legal notes>

legal notes
=================
| SPDX-FileCopyrightText: © 2022 ekvip automation GmbH <info@ekvip.de>
| SPDX-License-Identifier: Apache-2.0
| For details check: Apache-2.0_

.. _Apache-2.0: https://www.apache.org/licenses/LICENSE-2.0

.. </legal notes>



*)

METHOD msbIsEqualTo
VAR_INPUT
	(* current value to check *)
	currentValue	:WORD;
	(* expected value of msb *)
	expectedValue	:BOOL;
	(* message if the assertion is false *)
	message			:AssertMessage;
END_VAR
END_METHOD

(*

## Short summary
This assertion method checks if the most significant bit of current value
is not equal to the unexpected value

.. <legal notes>

legal notes
=================
| SPDX-FileCopyrightText: © 2022 ekvip automation GmbH <info@ekvip.de>
| SPDX-License-Identifier: Apache-2.0
| For details check: Apache-2.0_

.. _Apache-2.0: https://www.apache.org/licenses/LICENSE-2.0

.. </legal notes>



*)

METHOD msbIsNotEqualTo
VAR_INPUT
	(* current value to check *)
	currentValue	:WORD;
	(* unexpected value of msb *)
	unexpectedValue	:BOOL;
	(* message if the assertion is false *)
	message			:AssertMessage;
END_VAR
END_METHOD

(*

## Short summary
This assertion method checks if the most significant bit of current value
is set

.. <legal notes>

legal notes
=================
| SPDX-FileCopyrightText: © 2022 ekvip automation GmbH <info@ekvip.de>
| SPDX-License-Identifier: Apache-2.0
| For details check: Apache-2.0_

.. _Apache-2.0: https://www.apache.org/licenses/LICENSE-2.0

.. </legal notes>



*)

METHOD msbIsSet
VAR_INPUT
	(* current value to check *)
	currentValue	:WORD;
	(* message if the assertion is false *)
	message			:AssertMessage;
END_VAR
END_METHOD

(*

## Short summary
This assertion method checks if the most significant bit of current value
is unset

.. <legal notes>

legal notes
=================
| SPDX-FileCopyrightText: © 2022 ekvip automation GmbH <info@ekvip.de>
| SPDX-License-Identifier: Apache-2.0
| For details check: Apache-2.0_

.. _Apache-2.0: https://www.apache.org/licenses/LICENSE-2.0

.. </legal notes>



*)

METHOD msbIsUnset
VAR_INPUT
	(* current value to check *)
	currentValue	:WORD;
	(* message if the assertion is false *)
	message			:AssertMessage;
END_VAR
END_METHOD

(*

## Short summary
This assertion method checks if the result current value bitwise ``OR`` mask is equal to the expected value

.. <legal notes>

legal notes
=================
| SPDX-FileCopyrightText: © 2022 ekvip automation GmbH <info@ekvip.de>
| SPDX-License-Identifier: Apache-2.0
| For details check: Apache-2.0_

.. _Apache-2.0: https://www.apache.org/licenses/LICENSE-2.0

.. </legal notes>



*)

METHOD orMaskIsEqualTo
VAR_INPUT
	(* current value to check *)
	currentValue	:WORD;
	(* 2nd operand for bitwise operation *)
	mask			:WORD;
	(* expected result after masking *)
	expectedValue	:WORD;
	(* message if the assertion is false *)
	message			:AssertMessage;
END_VAR
END_METHOD

(*

## Short summary
This assertion method checks if the result current value bitwise ``OR`` mask 
is not equal to the unexpected value

.. <legal notes>

legal notes
=================
| SPDX-FileCopyrightText: © 2022 ekvip automation GmbH <info@ekvip.de>
| SPDX-License-Identifier: Apache-2.0
| For details check: Apache-2.0_

.. _Apache-2.0: https://www.apache.org/licenses/LICENSE-2.0

.. </legal notes>



*)

METHOD orMaskIsNotEqualTo
VAR_INPUT
	(* current value to check *)
	currentValue	:WORD;
	(* 2nd operand for bitwise operation *)
	mask			:WORD;
	(* unexpected result after masking *)
	unexpectedValue	:WORD;
	(* message if the assertion is false *)
	message			:AssertMessage;
END_VAR
END_METHOD

(*

## Short summary
This assertion method checks if the current value is equal to the expected value

.. <legal notes>

legal notes
=================
| SPDX-FileCopyrightText: © 2022 ekvip automation GmbH <info@ekvip.de>
| SPDX-License-Identifier: Apache-2.0
| For details check: Apache-2.0_

.. _Apache-2.0: https://www.apache.org/licenses/LICENSE-2.0

.. </legal notes>



*)

METHOD valueIsEqualTo
VAR_INPUT
	(* current value to check *)
	currentValue	:WORD;
	(* expected value to compare *)
	expectedValue	:WORD;
	(* message if the assertion is false *)
	message			:AssertMessage;
END_VAR
END_METHOD

(*

## Short summary
This assertion method checks if the current value is greater than the less value

.. <legal notes>

legal notes
=================
| SPDX-FileCopyrightText: © 2022 ekvip automation GmbH <info@ekvip.de>
| SPDX-License-Identifier: Apache-2.0
| For details check: Apache-2.0_

.. _Apache-2.0: https://www.apache.org/licenses/LICENSE-2.0

.. </legal notes>



*)

METHOD valueIsGreaterThan
VAR_INPUT
	(* current value to check *)
	currentValue	:WORD;
	(* less than lower limit *)
	lessValue		:WORD;
	(* message if the assertion is false *)
	message			:AssertMessage;
END_VAR
END_METHOD

(*

## Short summary
This assertion method checks if the current value is inside a limit

**Attention:** 
	limits are included: ``valueIsInRangeOf(3, 3, 3)`` is a true assertion

.. <legal notes>

legal notes
=================
| SPDX-FileCopyrightText: © 2022 ekvip automation GmbH <info@ekvip.de>
| SPDX-License-Identifier: Apache-2.0
| For details check: Apache-2.0_

.. _Apache-2.0: https://www.apache.org/licenses/LICENSE-2.0

.. </legal notes>



*)

METHOD valueIsInRangeOf
VAR_INPUT
	(* lower limit for the current value *)
	lowerLimit		:WORD;
	(* current value to check *)
	currentValue	:WORD;
	(* upper limit for the current value *)
	upperLimit		:WORD;
	(* message if the assertion is false *)
	message			:AssertMessage;
END_VAR
END_METHOD

(*

## Short summary
This assertion method checks if the current value is less than the greater value

.. <legal notes>

legal notes
=================
| SPDX-FileCopyrightText: © 2022 ekvip automation GmbH <info@ekvip.de>
| SPDX-License-Identifier: Apache-2.0
| For details check: Apache-2.0_

.. _Apache-2.0: https://www.apache.org/licenses/LICENSE-2.0

.. </legal notes>



*)

METHOD valueIsLessThan
VAR_INPUT
	(* current value to check *)
	currentValue	:WORD;
	(* greater than upper limit *)
	greaterValue	:WORD;
	(* message if the assertion is false *)
	message			:AssertMessage;
END_VAR
END_METHOD

(*

## Short summary
This assertion method checks if the current value is less than or equal to the maximum value

.. <legal notes>

legal notes
=================
| SPDX-FileCopyrightText: © 2022 ekvip automation GmbH <info@ekvip.de>
| SPDX-License-Identifier: Apache-2.0
| For details check: Apache-2.0_

.. _Apache-2.0: https://www.apache.org/licenses/LICENSE-2.0

.. </legal notes>



*)

METHOD valueIsMax
VAR_INPUT
	(* current value to check *)
	currentValue	:WORD;
	(* upper limit for the current value *)
	maximumValue	:WORD;
	(* message if the assertion is false *)
	message			:AssertMessage;
END_VAR
END_METHOD

(*

## Short summary
This assertion method checks if the current value is greater than or equal to the minimum value

.. <legal notes>

legal notes
=================
| SPDX-FileCopyrightText: © 2022 ekvip automation GmbH <info@ekvip.de>
| SPDX-License-Identifier: Apache-2.0
| For details check: Apache-2.0_

.. _Apache-2.0: https://www.apache.org/licenses/LICENSE-2.0

.. </legal notes>



*)

METHOD valueIsMin
VAR_INPUT
	(* current value to check *)
	currentValue	:WORD;
	(* lower limit for the current value *)
	minimumValue	:WORD;
	(* message if the assertion is false *)
	message			:AssertMessage;
END_VAR
END_METHOD

(*

## Short summary
This assertion method checks if the current value is not equal to the unexpected value

.. <legal notes>

legal notes
=================
| SPDX-FileCopyrightText: © 2022 ekvip automation GmbH <info@ekvip.de>
| SPDX-License-Identifier: Apache-2.0
| For details check: Apache-2.0_

.. _Apache-2.0: https://www.apache.org/licenses/LICENSE-2.0

.. </legal notes>



*)

METHOD valueIsNotEqualTo
VAR_INPUT
	(* current value to check *)
	currentValue	:WORD;
	(* unexpected value to compare *)
	unexpectedValue	:WORD;
	(* message if the assertion is false *)
	message			:AssertMessage;
END_VAR
END_METHOD

(*

## Short summary
This assertion method checks if the result current value bitwise ``XOR`` mask is equal to the expected value

.. <legal notes>

legal notes
=================
| SPDX-FileCopyrightText: © 2022 ekvip automation GmbH <info@ekvip.de>
| SPDX-License-Identifier: Apache-2.0
| For details check: Apache-2.0_

.. _Apache-2.0: https://www.apache.org/licenses/LICENSE-2.0

.. </legal notes>



*)

METHOD xorMaskIsEqualTo
VAR_INPUT
	(* current value to check *)
	currentValue	:WORD;
	(* 2nd operand for bitwise operation *)
	mask			:WORD;
	(* expected result after masking *)
	expectedValue	:WORD;
	(* message if the assertion is false *)
	message			:AssertMessage;
END_VAR
END_METHOD

(*

## Short summary
This assertion method checks if the result current value bitwise ``XOR`` mask 
is not equal to the unexpected value

.. <legal notes>

legal notes
=================
| SPDX-FileCopyrightText: © 2022 ekvip automation GmbH <info@ekvip.de>
| SPDX-License-Identifier: Apache-2.0
| For details check: Apache-2.0_

.. _Apache-2.0: https://www.apache.org/licenses/LICENSE-2.0

.. </legal notes>



*)

METHOD xorMaskIsNotEqualTo
VAR_INPUT
	(* current value to check *)
	currentValue	:WORD;
	(* 2nd operand for bitwise operation *)
	mask			:WORD;
	(* unexpected result after masking *)
	unexpectedValue	:WORD;
	(* message if the assertion is false *)
	message			:AssertMessage;
END_VAR
END_METHOD

END_INTERFACE

// ---- Assertor/Assertions/BitNumberAssertions/XWord/interfaces/IXWordAssertions.TcIO
(*

## Short summary
This interface provides assert statements for register length words  

.. <legal notes>

legal notes
=================
| SPDX-FileCopyrightText: © 2022 ekvip automation GmbH <info@ekvip.de>
| SPDX-License-Identifier: Apache-2.0
| For details check: Apache-2.0_

.. _Apache-2.0: https://www.apache.org/licenses/LICENSE-2.0

.. </legal notes>



*)

INTERFACE IXWordAssertions EXTENDS __SYSTEM.IQueryInterface

(*

## Short summary
This assertion method checks if the result current value bitwise ``AND`` mask is equal to the expected value

.. <legal notes>

legal notes
=================
| SPDX-FileCopyrightText: © 2022 ekvip automation GmbH <info@ekvip.de>
| SPDX-License-Identifier: Apache-2.0
| For details check: Apache-2.0_

.. _Apache-2.0: https://www.apache.org/licenses/LICENSE-2.0

.. </legal notes>



*)

METHOD andMaskIsEqualTo
VAR_INPUT
	(* current value to check *)
	currentValue	:__XWORD;
	(* 2nd operand for bitwise operation *)
	mask			:__XWORD;
	(* expected result after masking *)
	expectedValue	:__XWORD;
	(* message if the assertion is false *)
	message			:AssertMessage;
END_VAR
END_METHOD

(*

## Short summary
This assertion method checks if the result current value bitwise ``AND`` mask
is not equal to the unexpected value

.. <legal notes>

legal notes
=================
| SPDX-FileCopyrightText: © 2022 ekvip automation GmbH <info@ekvip.de>
| SPDX-License-Identifier: Apache-2.0
| For details check: Apache-2.0_

.. _Apache-2.0: https://www.apache.org/licenses/LICENSE-2.0

.. </legal notes>



*)

METHOD andMaskIsNotEqualTo
VAR_INPUT
	(* current value to check *)
	currentValue	:__XWORD;
	(* 2nd operand for bitwise operation *)
	mask			:__XWORD;
	(* unexpected result after masking *)
	unexpectedValue	:__XWORD;
	(* message if the assertion is false *)
	message			:AssertMessage;
END_VAR
END_METHOD

(*

## Short summary
This assertion method checks if the selected bit of current value
is equal to the expected value

.. <legal notes>

legal notes
=================
| SPDX-FileCopyrightText: © 2022 ekvip automation GmbH <info@ekvip.de>
| SPDX-License-Identifier: Apache-2.0
| For details check: Apache-2.0_

.. _Apache-2.0: https://www.apache.org/licenses/LICENSE-2.0

.. </legal notes>



*)

METHOD bitXIsEqualTo
VAR_INPUT
	(* current value to check *)
	currentValue	:__XWORD;
	(* number of bit to check *)
	number			:BitNumberXWord;	
	(* expected value of bit *)
	expectedValue	:BOOL;
	(* message if the assertion is false *)
	message			:AssertMessage;
END_VAR
END_METHOD

(*

## Short summary
This assertion method checks if the selected bit of current value
is not equal to the unexpected value

.. <legal notes>

legal notes
=================
| SPDX-FileCopyrightText: © 2022 ekvip automation GmbH <info@ekvip.de>
| SPDX-License-Identifier: Apache-2.0
| For details check: Apache-2.0_

.. _Apache-2.0: https://www.apache.org/licenses/LICENSE-2.0

.. </legal notes>



*)

METHOD bitXIsNotEqualTo
VAR_INPUT
	(* current value to check *)
	currentValue	:__XWORD;
	(* number of bit to check *)
	number			:BitNumberXWord;	
	(* unexpected value of bit *)
	unexpectedValue	:BOOL;
	(* message if the assertion is false *)
	message			:AssertMessage;
END_VAR
END_METHOD

(*

## Short summary
This assertion method checks if the selected bit of current value
is set

.. <legal notes>

legal notes
=================
| SPDX-FileCopyrightText: © 2022 ekvip automation GmbH <info@ekvip.de>
| SPDX-License-Identifier: Apache-2.0
| For details check: Apache-2.0_

.. _Apache-2.0: https://www.apache.org/licenses/LICENSE-2.0

.. </legal notes>



*)

METHOD bitXIsSet
VAR_INPUT
	(* current value to check *)
	currentValue	:__XWORD;
	(* number of bit to check *)
	number			:BitNumberXWord;	
	(* message if the assertion is false *)
	message			:AssertMessage;
END_VAR
END_METHOD

(*

## Short summary
This assertion method checks if the selected bit of current value
is unset

.. <legal notes>

legal notes
=================
| SPDX-FileCopyrightText: © 2022 ekvip automation GmbH <info@ekvip.de>
| SPDX-License-Identifier: Apache-2.0
| For details check: Apache-2.0_

.. _Apache-2.0: https://www.apache.org/licenses/LICENSE-2.0

.. </legal notes>



*)

METHOD bitXIsUnset
VAR_INPUT
	(* current value to check *)
	currentValue	:__XWORD;
	(* number of bit to check *)
	number			:BitNumberXWord;	
	(* message if the assertion is false *)
	message			:AssertMessage;
END_VAR
END_METHOD

(*

## Short summary
This assertion method checks if the least significant bit of current value
is equal to the expected value

.. <legal notes>

legal notes
=================
| SPDX-FileCopyrightText: © 2022 ekvip automation GmbH <info@ekvip.de>
| SPDX-License-Identifier: Apache-2.0
| For details check: Apache-2.0_

.. _Apache-2.0: https://www.apache.org/licenses/LICENSE-2.0

.. </legal notes>



*)

METHOD lsbIsEqualTo
VAR_INPUT
	(* current value to check *)
	currentValue	:__XWORD;
	(* expected value of lsb *)
	expectedValue	:BOOL;
	(* message if the assertion is false *)
	message			:AssertMessage;
END_VAR
END_METHOD

(*

## Short summary
This assertion method checks if the least significant bit of current value
is not equal to the unexpected value

.. <legal notes>

legal notes
=================
| SPDX-FileCopyrightText: © 2022 ekvip automation GmbH <info@ekvip.de>
| SPDX-License-Identifier: Apache-2.0
| For details check: Apache-2.0_

.. _Apache-2.0: https://www.apache.org/licenses/LICENSE-2.0

.. </legal notes>



*)

METHOD lsbIsNotEqualTo
VAR_INPUT
	(* current value to check *)
	currentValue	:__XWORD;
	(* unexpected value of lsb *)
	unexpectedValue	:BOOL;
	(* message if the assertion is false *)
	message			:AssertMessage;
END_VAR
END_METHOD

(*

## Short summary
This assertion method checks if the least significant bit of current value
is set

.. <legal notes>

legal notes
=================
| SPDX-FileCopyrightText: © 2022 ekvip automation GmbH <info@ekvip.de>
| SPDX-License-Identifier: Apache-2.0
| For details check: Apache-2.0_

.. _Apache-2.0: https://www.apache.org/licenses/LICENSE-2.0

.. </legal notes>



*)

METHOD lsbIsSet
VAR_INPUT
	(* current value to check *)
	currentValue	:__XWORD;
	(* message if the assertion is false *)
	message			:AssertMessage;
END_VAR
END_METHOD

(*

## Short summary
This assertion method checks if the least significant bit of current value
is unset

.. <legal notes>

legal notes
=================
| SPDX-FileCopyrightText: © 2022 ekvip automation GmbH <info@ekvip.de>
| SPDX-License-Identifier: Apache-2.0
| For details check: Apache-2.0_

.. _Apache-2.0: https://www.apache.org/licenses/LICENSE-2.0

.. </legal notes>



*)

METHOD lsbIsUnset
VAR_INPUT
	(* current value to check *)
	currentValue	:__XWORD;
	(* message if the assertion is false *)
	message			:AssertMessage;
END_VAR
END_METHOD

(*

## Short summary
This assertion method checks if the most significant bit of current value
is equal to the expected value

.. <legal notes>

legal notes
=================
| SPDX-FileCopyrightText: © 2022 ekvip automation GmbH <info@ekvip.de>
| SPDX-License-Identifier: Apache-2.0
| For details check: Apache-2.0_

.. _Apache-2.0: https://www.apache.org/licenses/LICENSE-2.0

.. </legal notes>



*)

METHOD msbIsEqualTo
VAR_INPUT
	(* current value to check *)
	currentValue	:__XWORD;
	(* expected value of msb *)
	expectedValue	:BOOL;
	(* message if the assertion is false *)
	message			:AssertMessage;
END_VAR
END_METHOD

(*

## Short summary
This assertion method checks if the most significant bit of current value
is not equal to the unexpected value

.. <legal notes>

legal notes
=================
| SPDX-FileCopyrightText: © 2022 ekvip automation GmbH <info@ekvip.de>
| SPDX-License-Identifier: Apache-2.0
| For details check: Apache-2.0_

.. _Apache-2.0: https://www.apache.org/licenses/LICENSE-2.0

.. </legal notes>



*)

METHOD msbIsNotEqualTo
VAR_INPUT
	(* current value to check *)
	currentValue	:__XWORD;
	(* unexpected value of msb *)
	unexpectedValue	:BOOL;
	(* message if the assertion is false *)
	message			:AssertMessage;
END_VAR
END_METHOD

(*

## Short summary
This assertion method checks if the most significant bit of current value
is set

.. <legal notes>

legal notes
=================
| SPDX-FileCopyrightText: © 2022 ekvip automation GmbH <info@ekvip.de>
| SPDX-License-Identifier: Apache-2.0
| For details check: Apache-2.0_

.. _Apache-2.0: https://www.apache.org/licenses/LICENSE-2.0

.. </legal notes>



*)

METHOD msbIsSet
VAR_INPUT
	(* current value to check *)
	currentValue	:__XWORD;
	(* message if the assertion is false *)
	message			:AssertMessage;
END_VAR
END_METHOD

(*

## Short summary
This assertion method checks if the most significant bit of current value
is unset

.. <legal notes>

legal notes
=================
| SPDX-FileCopyrightText: © 2022 ekvip automation GmbH <info@ekvip.de>
| SPDX-License-Identifier: Apache-2.0
| For details check: Apache-2.0_

.. _Apache-2.0: https://www.apache.org/licenses/LICENSE-2.0

.. </legal notes>



*)

METHOD msbIsUnset
VAR_INPUT
	(* current value to check *)
	currentValue	:__XWORD;
	(* message if the assertion is false *)
	message			:AssertMessage;
END_VAR
END_METHOD

(*

## Short summary
This assertion method checks if the result current value bitwise ``OR`` mask is equal to the expected value

.. <legal notes>

